   1:  PR[91,2] = PR[90,2] + 16.760;
   1:L PR[91] R[100]mm/sec CNT100;
   1:  PR[91,1] = PR[90,1] + -20.956;
   1:  PR[91,2] = PR[90,2] + 17.044;
   1:L PR[91] R[100]mm/sec CNT100;
   1:  PR[91,1] = PR[90,1] + -22.141;
   1:  PR[91,2] = PR[90,2] + 17.148;
   1:L PR[91] R[100]mm/sec CNT100;
   1:  PR[91,1] = PR[90,1] + -24.744;
   1:  PR[91,2] = PR[90,2] + 17.432;
   1:L PR[91] R[100]mm/sec CNT100;
   1:  PR[91,1] = PR[90,1] + -25.936;
   1:  PR[91,2] = PR[90,2] + 17.327;
   1:L PR[91] R[100]mm/sec CNT100;
   1:  PR[91,1] = PR[90,1] + -28.415;
   1:  PR[91,2] = PR[90,2] + 17.040;
   1:L PR[91] R[100]mm/sec CNT100;
   1:  PR[91,1] = PR[90,1] + -29.641;
   1:  PR[91,2] = PR[90,2] + 16.711;
   1:L PR[91] R[100]mm/sec CNT100;
   1:  PR[91,1] = PR[90,1] + -31.889;
   1:  PR[91,2] = PR[90,2] + 15.918;
   1:L PR[91] R[100]mm/sec CNT100;
   1:  PR[91,1] = PR[90,1] + -33.097;
   1:  PR[91,2] = PR[90,2] + 15.354;
   1:L PR[91] R[100]mm/sec CNT100;
   1:  PR[91,1] = PR[90,1] + -35.033;
   1:  PR[91,2] = PR[90,2] + 14.131;
   1:L PR[91] R[100]mm/sec CNT100;
   1:  PR[91,1] = PR[90,1] + -36.169;
   1:  PR[91,2] = PR[90,2] + 13.336;
   1:L PR[91] R[100]mm/sec CNT100;
   1:  PR[91,1] = PR[90,1] + -38.779;
   1:  PR[91,2] = PR[90,2] + 10.719;
   1:L PR[91] R[100]mm/sec CNT100TB   .50sec,CALL END_PUD;
   1:  PR[92] = PR[91];
   1:  PR[92,3] = PR[92,3] + 20;
   1:J PR[92] 10% FINE;
   1:  PR[91,1] = PR[90,1] + -69.247;
   1:  PR[91,2] = PR[90,2] + 16.551;
   1:  PR[92] = PR[91];
   1:  PR[92,3] = PR[92,3] + 20;
   1:J PR[92] 10% FINE;
   1:L PR[91] R[100]mm/sec CNT100;
   1:  CALL LASER_DRAHT_START;
   1:  PR[91,1] = PR[90,1] + -72.638;
   1:  PR[91,2] = PR[90,2] + 17.266;
   1:L PR[91] R[100]mm/sec CNT100;
   1:  PR[91,1] = PR[90,1] + -73.009;
   1:  PR[91,2] = PR[90,2] + 17.298;
   1:L PR[91] R[100]mm/sec CNT100;
   1:  PR[91,1] = PR[90,1] + -76.253;
   1:  PR[91,2] = PR[90,2] + 17.293;
   1:L PR[91] R[100]mm/sec CNT100;
   1:  PR[91,1] = PR[90,1] + -76.771;
   1:  PR[91,2] = PR[90,2] + 17.248;
   1:L PR[91] R[100]mm/sec CNT100;
   1:  PR[91,1] = PR[90,1] + -79.751;
   1:  PR[91,2] = PR[90,2] + 16.609;
   1:L PR[91] R[100]mm/sec CNT100;
   1:  PR[91,1] = PR[90,1] + -80.365;
   1:  PR[91,2] = PR[90,2] + 16.445;
   1:L PR[91] R[100]mm/sec CNT100;
   1:  PR[91,1] = PR[90,1] + -81.001;
   1:  PR[91,2] = PR[90,2] + 16.148;
   1:L PR[91] R[100]mm/sec CNT100;
   1:  PR[91,1] = PR[90,1] + -83.731;
   1:  PR[91,2] = PR[90,2] + 14.925;
   1:L PR[91] R[100]mm/sec CNT100;
   1:  PR[91,1] = PR[90,1] + -84.359;
   1:  PR[91,2] = PR[90,2] + 14.485;
   1:L PR[91] R[100]mm/sec CNT100;
   1:  PR[91,1] = PR[90,1] + -86.653;
   1:  PR[91,2] = PR[90,2] + 12.813;
   1:L PR[91] R[100]mm/sec CNT100;
   1:  PR[91,1] = PR[90,1] + -87.257;
   1:  PR[91,2] = PR[90,2] + 12.209;
   1:L PR[91] R[100]mm/sec CNT100;
   1:  PR[91,1] = PR[90,1] + -89.073;
   1:  PR[91,2] = PR[90,2] + 10.188;
   1:L PR[91] R[100]mm/sec CNT100;
   1:  PR[91,1] = PR[90,1] + -89.607;
   1:  PR[91,2] = PR[90,2] + 9.426;
   1:L PR[91] R[100]mm/sec CNT100;
   1:  PR[91,1] = PR[90,1] + -90.920;
   1:  PR[91,2] = PR[90,2] + 7.148;
   1:L PR[91] R[100]mm/sec CNT100;
   1:  PR[91,1] = PR[90,1] + -91.333;
   1:  PR[91,2] = PR[90,2] + 6.263;
   1:L PR[91] R[100]mm/sec CNT100;
   1:  PR[91,1] = PR[90,1] + -92.127;
   1:  PR[91,2] = PR[90,2] + 3.815;
   1:L PR[91] R[100]mm/sec CNT100;
   1:  PR[91,1] = PR[90,1] + -92.384;
   1:  PR[91,2] = PR[90,2] + 2.855;
   1:L PR[91] R[100]mm/sec CNT100;
   1:  PR[91,1] = PR[90,1] + -92.476;
   1:  PR[91,2] = PR[90,2] + 1.801;
   1:L PR[91] R[100]mm/sec CNT100;
   1:  PR[91,1] = PR[90,1] + -92.743;
   1:  PR[91,2] = PR[90,2] + -0.747;
   1:L PR[91] R[100]mm/sec CNT100;
   1:  PR[91,1] = PR[90,1] + -92.665;
   1:  PR[91,2] = PR[90,2] + -1.630;
   1:L PR[91] R[100]mm/sec CNT100;
   1:  PR[91,1] = PR[90,1] + -92.614;
   1:  PR[91,2] = PR[90,2] + -1.837;
   1:L PR[91] R[100]mm/sec CNT100;
   1:  PR[91,1] = PR[90,1] + -92.361;
   1:  PR[91,2] = PR[90,2] + -4.254;
   1:L PR[91] R[100]mm/sec CNT100;
   1:  PR[91,1] = PR[90,1] + -92.040;
   1:  PR[91,2] = PR[90,2] + -5.451;
   1:L PR[91] R[100]mm/sec CNT100;
   1:  PR[91,1] = PR[90,1] + -91.331;
   1:  PR[91,2] = PR[90,2] + -7.640;
   1:L PR[91] R[100]mm/sec CNT100;
   1:  PR[91,1] = PR[90,1] + -90.820;
   1:  PR[91,2] = PR[90,2] + -8.736;
   1:L PR[91] R[100]mm/sec CNT100;
   1:  PR[91,1] = PR[90,1] + -89.646;
   1:  PR[91,2] = PR[90,2] + -10.772;
   1:L PR[91] R[100]mm/sec CNT100;
   1:  PR[91,1] = PR[90,1] + -88.976;
   1:  PR[91,2] = PR[90,2] + -11.729;
   1:L PR[91] R[100]mm/sec CNT100;
   1:  PR[91,1] = PR[90,1] + -87.353;
   1:  PR[91,2] = PR[90,2] + -13.536;
   1:L PR[91] R[100]mm/sec CNT100;
   1:  PR[91,1] = PR[90,1] + -86.576;
   1:  PR[91,2] = PR[90,2] + -14.313;
   1:L PR[91] R[100]mm/sec CNT100;
   1:  PR[91,1] = PR[90,1] + -84.525;
   1:  PR[91,2] = PR[90,2] + -15.809;
   1:L PR[91] R[100]mm/sec CNT100;
   1:  PR[91,1] = PR[90,1] + -83.677;
   1:  PR[91,2] = PR[90,2] + -16.402;
   1:L PR[91] R[100]mm/sec CNT100;
   1:  PR[91,1] = PR[90,1] + -82.739;
   1:  PR[91,2] = PR[90,2] + -16.839;
   1:L PR[91] R[100]mm/sec CNT100;
   1:  PR[91,1] = PR[90,1] + -80.387;
   1:  PR[91,2] = PR[90,2] + -17.893;
   1:L PR[91] R[100]mm/sec CNT100;
   1:  PR[91,1] = PR[90,1] + -79.501;
   1:  PR[91,2] = PR[90,2] + -18.130;
   1:L PR[91] R[100]mm/sec CNT100;
   1:  PR[91,1] = PR[90,1] + -76.834;
   1:  PR[91,2] = PR[90,2] + -18.703;
   1:L PR[91] R[100]mm/sec CNT100;
   1:  PR[91,1] = PR[90,1] + -76.040;
   1:  PR[91,2] = PR[90,2] + -18.772;
   1:L PR[91] R[100]mm/sec CNT100;
   1:  PR[91,1] = PR[90,1] + -73.135;
   1:  PR[91,2] = PR[90,2] + -18.779;
   1:L PR[91] R[100]mm/sec CNT100;
   1:  PR[91,1] = PR[90,1] + -72.474;
   1:  PR[91,2] = PR[90,2] + -18.721;
   1:L PR[91] R[100]mm/sec CNT100;
   1:  PR[91,1] = PR[90,1] + -69.435;
   1:  PR[91,2] = PR[90,2] + -18.082;
   1:L PR[91] R[100]mm/sec CNT100;
   1:  PR[91,1] = PR[90,1] + -68.955;
   1:  PR[91,2] = PR[90,2] + -17.954;
   1:L PR[91] R[100]mm/sec CNT100;
   1:  PR[91,1] = PR[90,1] + -68.437;
   1:  PR[91,2] = PR[90,2] + -17.712;
   1:L PR[91] R[100]mm/sec CNT100;
   1:  PR[91,1] = PR[90,1] + -65.552;
   1:  PR[91,2] = PR[90,2] + -16.440;
   1:L PR[91] R[100]mm/sec CNT100;
   1:  PR[91,1] = PR[90,1] + -62.499;
   1:  PR[91,2] = PR[90,2] + -14.245;
   1:L PR[91] R[100]mm/sec CNT100;
   1:  PR[91,1] = PR[90,1] + -62.350;
   1:  PR[91,2] = PR[90,2] + -14.095;
   1:L PR[91] R[100]mm/sec CNT100;
   1:  PR[91,1] = PR[90,1] + -59.945;
   1:  PR[91,2] = PR[90,2] + -11.434;
   1:L PR[91] R[100]mm/sec CNT100;
   1:  PR[91,1] = PR[90,1] + -59.899;
   1:  PR[91,2] = PR[90,2] + -11.367;
   1:L PR[91] R[100]mm/sec CNT100;
   1:  PR[91,1] = PR[90,1] + -58.021;
   1:  PR[91,2] = PR[90,2] + -8.128;
   1:L PR[91] R[100]mm/sec CNT100;
   1:  PR[91,1] = PR[90,1] + -56.846;
   1:  PR[91,2] = PR[90,2] + -4.503;
   1:L PR[91] R[100]mm/sec CNT100;
   1:  PR[91,1] = PR[90,1] + -56.756;
   1:  PR[91,2] = PR[90,2] + -3.498;
   1:L PR[91] R[100]mm/sec CNT100;
   1:  PR[91,1] = PR[90,1] + -56.459;
   1:  PR[91,2] = PR[90,2] + -0.724;
   1:L PR[91] R[100]mm/sec CNT100;
   1:  PR[91,1] = PR[90,1] + -56.811;
   1:  PR[91,2] = PR[90,2] + 2.748;
   1:L PR[91] R[100]mm/sec CNT100;
   1:  PR[91,1] = PR[90,1] + -56.836;
   1:  PR[91,2] = PR[90,2] + 3.070;
   1:L PR[91] R[100]mm/sec CNT100;
   1:  PR[91,1] = PR[90,1] + -58.024;
   1:  PR[91,2] = PR[90,2] + 6.648;
   1:L PR[91] R[100]mm/sec CNT100;
   1:  PR[91,1] = PR[90,1] + -59.962;
   1:  PR[91,2] = PR[90,2] + 9.930;
   1:L PR[91] R[100]mm/sec CNT100;
   1:  PR[91,1] = PR[90,1] + -62.542;
   1:  PR[91,2] = PR[90,2] + 12.758;
   1:L PR[91] R[100]mm/sec CNT100;
   1:  PR[91,1] = PR[90,1] + -65.608;
   1:  PR[91,2] = PR[90,2] + 14.970;
   1:L PR[91] R[100]mm/sec CNT100;
   1:  PR[91,1] = PR[90,1] + -69.045;
   1:  PR[91,2] = PR[90,2] + 16.497;
   1:L PR[91] R[100]mm/sec CNT100;
   1:  PR[91,1] = PR[90,1] + -69.247;
   1:  PR[91,2] = PR[90,2] + 16.551;
   1:L PR[91] R[100]mm/sec CNT100TB   .50sec,CALL END_PUD;
   1:  PR[92] = PR[91];
   1:  PR[92,3] = PR[92,3] + 20;
   1:J PR[92] 10% FINE;
   1:  PR[91] = PR[90];
   1:  PR[91,1] = PR[90,1] + 39.926;
   1:  PR[91,2] = PR[90,2] + -10.972;
   1:  PR[91,3] = PR[90,3] + 17.095;
   1:  PR[92] = PR[91];
   1:  PR[92,3] = PR[92,3] + 20;
   1:J PR[92] 10% FINE;
   1:L PR[91] R[100]mm/sec CNT100;
   1:  CALL LASER_DRAHT_START;
   1:  PR[91,1] = PR[90,1] + 40.681;
   1:  PR[91,2] = PR[90,2] + -9.894;
   1:L PR[91] R[100]mm/sec CNT100;
   1:  PR[91,1] = PR[90,1] + 41.235;
   1:  PR[91,2] = PR[90,2] + -8.707;
   1:L PR[91] R[100]mm/sec CNT100;
   1:  PR[91,1] = PR[90,1] + 42.319;
   1:  PR[91,2] = PR[90,2] + -6.084;
   1:L PR[91] R[100]mm/sec CNT100;
   1:  PR[91,1] = PR[90,1] + 42.639;
   1:  PR[91,2] = PR[90,2] + -4.891;
   1:L PR[91] R[100]mm/sec CNT100;
   1:  PR[91,1] = PR[90,1] + 42.760;
   1:  PR[91,2] = PR[90,2] + -3.506;
   1:L PR[91] R[100]mm/sec CNT100;
   1:  PR[91,1] = PR[90,1] + 43.087;
   1:  PR[91,2] = PR[90,2] + -0.700;
   1:L PR[91] R[100]mm/sec CNT100;
   1:  PR[91,1] = PR[90,1] + 43.018;
   1:  PR[91,2] = PR[90,2] + 0.088;
   1:L PR[91] R[100]mm/sec CNT100;
   1:  PR[91,1] = PR[90,1] + 43.010;
   1:  PR[91,2] = PR[90,2] + 0.654;
   1:L PR[91] R[100]mm/sec CNT100;
   1:  PR[91,1] = PR[90,1] + 42.650;
   1:  PR[91,2] = PR[90,2] + 3.390;
   1:L PR[91] R[100]mm/sec CNT100;
   1:  PR[91,1] = PR[90,1] + 42.319;
   1:  PR[91,2] = PR[90,2] + 4.626;
   1:L PR[91] R[100]mm/sec CNT100;
   1:  PR[91,1] = PR[90,1] + 41.234;
   1:  PR[91,2] = PR[90,2] + 7.249;
   1:L PR[91] R[100]mm/sec CNT100;
   1:  PR[91,1] = PR[90,1] + 40.680;
   1:  PR[91,2] = PR[90,2] + 8.436;
   1:L PR[91] R[100]mm/sec CNT100;
   1:  PR[91,1] = PR[90,1] + 39.925;
   1:  PR[91,2] = PR[90,2] + 9.514;
   1:L PR[91] R[100]mm/sec CNT100;
   1:  PR[91,1] = PR[90,1] + 38.193;
   1:  PR[91,2] = PR[90,2] + 11.777;
   1:L PR[91] R[100]mm/sec CNT100;
   1:  PR[91,1] = PR[90,1] + 37.306;
   1:  PR[91,2] = PR[90,2] + 12.663;
   1:L PR[91] R[100]mm/sec CNT100;
   1:  PR[91,1] = PR[90,1] + 35.023;
   1:  PR[91,2] = PR[90,2] + 14.420;
   1:L PR[91] R[100]mm/sec CNT100;
   1:  PR[91,1] = PR[90,1] + 33.972;
   1:  PR[91,2] = PR[90,2] + 15.155;
   1:L PR[91] R[100]mm/sec CNT100;
   1:  PR[91,1] = PR[90,1] + 32.809;
   1:  PR[91,2] = PR[90,2] + 15.697;
   1:L PR[91] R[100]mm/sec CNT100;
   1:  PR[91,1] = PR[90,1] + 30.132;
   1:  PR[91,2] = PR[90,2] + 16.810;
   1:L PR[91] R[100]mm/sec CNT100;
   1:  PR[91,1] = PR[90,1] + 28.953;
   1:  PR[91,2] = PR[90,2] + 17.126;
   1:L PR[91] R[100]mm/sec CNT100;
   1:  PR[91,1] = PR[90,1] + 26.036;
   1:  PR[91,2] = PR[90,2] + 17.515;
   1:L PR[91] R[100]mm/sec CNT100;
   1:  PR[91,1] = PR[90,1] + 24.803;
   1:  PR[91,2] = PR[90,2] + 17.623;
   1:L PR[91] R[100]mm/sec CNT100;
   1:  PR[91,1] = PR[90,1] + 23.566;
   1:  PR[91,2] = PR[90,2] + 17.514;
   1:L PR[91] R[100]mm/sec CNT100;
   1:  PR[91,1] = PR[90,1] + 20.624;
   1:  PR[91,2] = PR[90,2] + 17.131;
   1:L PR[91] R[100]mm/sec CNT100;
   1:  PR[91,1] = PR[90,1] + 19.533;
   1:  PR[91,2] = PR[90,2] + 16.839;
   1:L PR[91] R[100]mm/sec CNT100;
   1:  PR[91,1] = PR[90,1] + 18.350;
   1:  PR[91,2] = PR[90,2] + 16.287;
   1:L PR[91] R[100]mm/sec CNT100;
   1:  PR[91,1] = PR[90,1] + 15.586;
   1:  PR[91,2] = PR[90,2] + 15.148;
   1:L PR[91] R[100]mm/sec CNT100;
   1:  PR[91,1] = PR[90,1] + 14.640;
   1:  PR[91,2] = PR[90,2] + 14.486;
   1:L PR[91] R[100]mm/sec CNT100;
   1:  PR[91,1] = PR[90,1] + 12.231;
   1:  PR[91,2] = PR[90,2] + 12.643;
   1:L PR[91] R[100]mm/sec CNT100;
   1:  PR[91,1] = PR[90,1] + 11.430;
   1:  PR[91,2] = PR[90,2] + 11.843;
   1:L PR[91] R[100]mm/sec CNT100;
   1:  PR[91,1] = PR[90,1] + 9.561;
   1:  PR[91,2] = PR[90,2] + 9.411;
   1:L PR[91] R[100]mm/sec CNT100;
   1:  PR[91,1] = PR[90,1] + 8.892;
   1:  PR[91,2] = PR[90,2] + 8.456;
   1:L PR[91] R[100]mm/sec CNT100;
   1:  PR[91,1] = PR[90,1] + 8.401;
   1:  PR[91,2] = PR[90,2] + 7.402;
   1:L PR[91] R[100]mm/sec CNT100;
   1:  PR[91,1] = PR[90,1] + 7.220;
   1:  PR[91,2] = PR[90,2] + 4.557;
   1:L PR[91] R[100]mm/sec CNT100;
   1:  PR[91,1] = PR[90,1] + 6.944;
   1:  PR[91,2] = PR[90,2] + 3.525;
   1:L PR[91] R[100]mm/sec CNT100;
   1:  PR[91,1] = PR[90,1] + 6.836;
   1:  PR[91,2] = PR[90,2] + 2.291;
   1:L PR[91] R[100]mm/sec CNT100;
   1:  PR[91,1] = PR[90,1] + 6.437;
   1:  PR[91,2] = PR[90,2] + -0.772;
   1:L PR[91] R[100]mm/sec CNT100;
   1:  PR[91,1] = PR[90,1] + 6.545;
   1:  PR[91,2] = PR[90,2] + -2.003;
   1:L PR[91] R[100]mm/sec CNT100;
   1:  PR[91,1] = PR[90,1] + 6.932;
   1:  PR[91,2] = PR[90,2] + -4.941;
   1:L PR[91] R[100]mm/sec CNT100;
   1:  PR[91,1] = PR[90,1] + 7.221;
   1:  PR[91,2] = PR[90,2] + -6.017;
   1:L PR[91] R[100]mm/sec CNT100;
   1:  PR[91,1] = PR[90,1] + 8.401;
   1:  PR[91,2] = PR[90,2] + -8.861;
   1:L PR[91] R[100]mm/sec CNT100;
   1:  PR[91,1] = PR[90,1] + 8.893;
   1:  PR[91,2] = PR[90,2] + -9.916;
   1:L PR[91] R[100]mm/sec CNT100;
   1:  PR[91,1] = PR[90,1] + 9.562;
   1:  PR[91,2] = PR[90,2] + -10.871;
   1:L PR[91] R[100]mm/sec CNT100;
   1:  PR[91,1] = PR[90,1] + 11.432;
   1:  PR[91,2] = PR[90,2] + -13.303;
   1:L PR[91] R[100]mm/sec CNT100;
   1:  PR[91,1] = PR[90,1] + 12.233;
   1:  PR[91,2] = PR[90,2] + -14.104;
   1:L PR[91] R[100]mm/sec CNT100;
   1:  PR[91,1] = PR[90,1] + 14.642;
   1:  PR[91,2] = PR[90,2] + -15.947;
   1:L PR[91] R[100]mm/sec CNT100;
   1:  PR[91,1] = PR[90,1] + 15.626;
   1:  PR[91,2] = PR[90,2] + -16.635;
   1:L PR[91] R[100]mm/sec CNT100;
   1:  PR[91,1] = PR[90,1] + 16.708;
   1:  PR[91,2] = PR[90,2] + -17.139;
   1:L PR[91] R[100]mm/sec CNT100;
   1:  PR[91,1] = PR[90,1] + 19.492;
   1:  PR[91,2] = PR[90,2] + -18.287;
   1:L PR[91] R[100]mm/sec CNT100;
   1:  PR[91,1] = PR[90,1] + 20.629;
   1:  PR[91,2] = PR[90,2] + -18.591;
   1:L PR[91] R[100]mm/sec CNT100;
   1:  PR[91,1] = PR[90,1] + 23.571;
   1:  PR[91,2] = PR[90,2] + -18.974;
   1:L PR[91] R[100]mm/sec CNT100;
   1:  PR[91,1] = PR[90,1] + 24.807;
   1:  PR[91,2] = PR[90,2] + -19.082;
   1:L PR[91] R[100]mm/sec CNT100;
   1:  PR[91,1] = PR[90,1] + 26.041;
   1:  PR[91,2] = PR[90,2] + -18.973;
   1:L PR[91] R[100]mm/sec CNT100;
   1:  PR[91,1] = PR[90,1] + 28.958;
   1:  PR[91,2] = PR[90,2] + -18.584;
   1:L PR[91] R[100]mm/sec CNT100;
   1:  PR[91,1] = PR[90,1] + 30.095;
   1:  PR[91,2] = PR[90,2] + -18.279;
   1:L PR[91] R[100]mm/sec CNT100;
   1:  PR[91,1] = PR[90,1] + 31.314;
   1:  PR[91,2] = PR[90,2] + -17.710;
   1:L PR[91] R[100]mm/sec CNT100;
   1:  PR[91,1] = PR[90,1] + 34.009;
   1:  PR[91,2] = PR[90,2] + -16.588;
   1:L PR[91] R[100]mm/sec CNT100;
   1:  PR[91,1] = PR[90,1] + 35.025;
   1:  PR[91,2] = PR[90,2] + -15.877;
   1:L PR[91] R[100]mm/sec CNT100;
   1:  PR[91,1] = PR[90,1] + 37.309;
   1:  PR[91,2] = PR[90,2] + -14.120;
   1:L PR[91] R[100]mm/sec CNT100;
   1:  PR[91,1] = PR[90,1] + 38.194;
   1:  PR[91,2] = PR[90,2] + -13.235;
   1:L PR[91] R[100]mm/sec CNT100;
   1:  PR[91,1] = PR[90,1] + 39.926;
   1:  PR[91,2] = PR[90,2] + -10.972;
   1:L PR[91] R[100]mm/sec CNT100TB   .50sec,CALL END_PUD;
   1:  PR[92] = PR[91];
   1:  PR[92,3] = PR[92,3] + 20;
   1:J PR[92] 10% FINE;
   1:  PR[91,1] = PR[90,1] + 66.363;
   1:  PR[91,2] = PR[90,2] + -17.228;
   1:  PR[92] = PR[91];
   1:  PR[92,3] = PR[92,3] + 20;
   1:J PR[92] 10% FINE;
   1:L PR[91] R[100]mm/sec CNT100;
   1:  CALL LASER_DRAHT_START;
   1:  PR[91,1] = PR[90,1] + 70.322;
   1:  PR[91,2] = PR[90,2] + -18.536;
   1:L PR[91] R[100]mm/sec CNT100;
   1:  PR[91,1] = PR[90,1] + 74.437;
   1:  PR[91,2] = PR[90,2] + -18.969;
   1:L PR[91] R[100]mm/sec CNT100;
   1:  PR[91,1] = PR[90,1] + 78.453;
   1:  PR[91,2] = PR[90,2] + -18.498;
   1:L PR[91] R[100]mm/sec CNT100;
   1:  PR[91,1] = PR[90,1] + 78.574;
   1:  PR[91,2] = PR[90,2] + -18.466;
   1:L PR[91] R[100]mm/sec CNT100;
   1:  PR[91,1] = PR[90,1] + 82.168;
   1:  PR[91,2] = PR[90,2] + -17.196;
   1:L PR[91] R[100]mm/sec CNT100;
   1:  PR[91,1] = PR[90,1] + 82.426;
   1:  PR[91,2] = PR[90,2] + -17.075;
   1:L PR[91] R[100]mm/sec CNT100;
   1:  PR[91,1] = PR[90,1] + 85.451;
   1:  PR[91,2] = PR[90,2] + -15.161;
   1:L PR[91] R[100]mm/sec CNT100;
   1:  PR[91,1] = PR[90,1] + 85.794;
   1:  PR[91,2] = PR[90,2] + -14.921;
   1:L PR[91] R[100]mm/sec CNT100;
   1:  PR[91,1] = PR[90,1] + 88.596;
   1:  PR[91,2] = PR[90,2] + -12.106;
   1:L PR[91] R[100]mm/sec CNT100;
   1:  PR[91,1] = PR[90,1] + 88.895;
   1:  PR[91,2] = PR[90,2] + -11.679;
   1:L PR[91] R[100]mm/sec CNT100;
   1:  PR[91,1] = PR[90,1] + 90.676;
   1:  PR[91,2] = PR[90,2] + -8.834;
   1:L PR[91] R[100]mm/sec CNT100;
   1:  PR[91,1] = PR[90,1] + 90.926;
   1:  PR[91,2] = PR[90,2] + -8.298;
   1:L PR[91] R[100]mm/sec CNT100;
   1:  PR[91,1] = PR[90,1] + 91.999;
   1:  PR[91,2] = PR[90,2] + -5.217;
   1:L PR[91] R[100]mm/sec CNT100;
   1:  PR[91,1] = PR[90,1] + 92.158;
   1:  PR[91,2] = PR[90,2] + -4.626;
   1:L PR[91] R[100]mm/sec CNT100;
   1:  PR[91,1] = PR[90,1] + 92.219;
   1:  PR[91,2] = PR[90,2] + -3.924;
   1:L PR[91] R[100]mm/sec CNT100;
   1:  PR[91,1] = PR[90,1] + 92.576;
   1:  PR[91,2] = PR[90,2] + -0.706;
   1:L PR[91] R[100]mm/sec CNT100;
   1:  PR[91,1] = PR[90,1] + 92.516;
   1:  PR[91,2] = PR[90,2] + -0.019;
   1:L PR[91] R[100]mm/sec CNT100;
   1:  PR[91,1] = PR[90,1] + 92.164;
   1:  PR[91,2] = PR[90,2] + 3.145;
   1:L PR[91] R[100]mm/sec CNT100;
   1:  PR[91,1] = PR[90,1] + 92.000;
   1:  PR[91,2] = PR[90,2] + 3.757;
   1:L PR[91] R[100]mm/sec CNT100;
   1:  PR[91,1] = PR[90,1] + 90.926;
   1:  PR[91,2] = PR[90,2] + 6.839;
   1:L PR[91] R[100]mm/sec CNT100;
   1:  PR[91,1] = PR[90,1] + 90.676;
   1:  PR[91,2] = PR[90,2] + 7.374;
   1:L PR[91] R[100]mm/sec CNT100;
   1:  PR[91,1] = PR[90,1] + 88.895;
   1:  PR[91,2] = PR[90,2] + 10.220;
   1:L PR[91] R[100]mm/sec CNT100;
   1:  PR[91,1] = PR[90,1] + 88.596;
   1:  PR[91,2] = PR[90,2] + 10.646;
   1:L PR[91] R[100]mm/sec CNT100;
   1:  PR[91,1] = PR[90,1] + 85.795;
   1:  PR[91,2] = PR[90,2] + 13.461;
   1:L PR[91] R[100]mm/sec CNT100;
   1:  PR[91,1] = PR[90,1] + 85.452;
   1:  PR[91,2] = PR[90,2] + 13.702;
   1:L PR[91] R[100]mm/sec CNT100;
   1:  PR[91,1] = PR[90,1] + 82.427;
   1:  PR[91,2] = PR[90,2] + 15.616;
   1:L PR[91] R[100]mm/sec CNT100;
   1:  PR[91,1] = PR[90,1] + 82.169;
   1:  PR[91,2] = PR[90,2] + 15.736;
   1:L PR[91] R[100]mm/sec CNT100;
   1:  PR[91,1] = PR[90,1] + 78.575;
   1:  PR[91,2] = PR[90,2] + 17.007;
   1:L PR[91] R[100]mm/sec CNT100;
   1:  PR[91,1] = PR[90,1] + 78.454;
   1:  PR[91,2] = PR[90,2] + 17.039;
   1:L PR[91] R[100]mm/sec CNT100;
   1:  PR[91,1] = PR[90,1] + 74.404;
   1:  PR[91,2] = PR[90,2] + 17.509;
   1:L PR[91] R[100]mm/sec CNT100;
   1:  PR[91,1] = PR[90,1] + 70.322;
   1:  PR[91,2] = PR[90,2] + 17.077;
   1:L PR[91] R[100]mm/sec CNT100;
   1:  PR[91,1] = PR[90,1] + 66.363;
   1:  PR[91,2] = PR[90,2] + 15.770;
   1:L PR[91] R[100]mm/sec CNT100;
   1:  PR[91,1] = PR[90,1] + 62.797;
   1:  PR[91,2] = PR[90,2] + 13.627;
   1:L PR[91] R[100]mm/sec CNT100;
   1:  PR[91,1] = PR[90,1] + 60.309;
   1:  PR[91,2] = PR[90,2] + 11.224;
   1:L PR[91] R[100]mm/sec CNT100;
   1:  PR[91,1] = PR[90,1] + 59.790;
   1:  PR[91,2] = PR[90,2] + 10.737;
   1:L PR[91] R[100]mm/sec CNT100;
   1:  PR[91,1] = PR[90,1] + 57.527;
   1:  PR[91,2] = PR[90,2] + 7.273;
   1:L PR[91] R[100]mm/sec CNT100;
   1:  PR[91,1] = PR[90,1] + 56.112;
   1:  PR[91,2] = PR[90,2] + 3.380;
   1:L PR[91] R[100]mm/sec CNT100;
   1:  PR[91,1] = PR[90,1] + 55.793;
   1:  PR[91,2] = PR[90,2] + 0.666;
   1:L PR[91] R[100]mm/sec CNT100;
   1:  PR[91,1] = PR[90,1] + 55.791;
   1:  PR[91,2] = PR[90,2] + 0.069;
   1:L PR[91] R[100]mm/sec CNT100;
   1:  PR[91,1] = PR[90,1] + 55.695;
   1:  PR[91,2] = PR[90,2] + -0.750;
   1:L PR[91] R[100]mm/sec CNT100;
   1:  PR[91,1] = PR[90,1] + 55.965;
   1:  PR[91,2] = PR[90,2] + -3.567;
   1:L PR[91] R[100]mm/sec CNT100;
   1:  PR[91,1] = PR[90,1] + 56.113;
   1:  PR[91,2] = PR[90,2] + -4.840;
   1:L PR[91] R[100]mm/sec CNT100;
   1:  PR[91,1] = PR[90,1] + 57.527;
   1:  PR[91,2] = PR[90,2] + -8.732;
   1:L PR[91] R[100]mm/sec CNT100;
   1:  PR[91,1] = PR[90,1] + 59.798;
   1:  PR[91,2] = PR[90,2] + -12.207;
   1:L PR[91] R[100]mm/sec CNT100;
   1:  PR[91,1] = PR[90,1] + 62.356;
   1:  PR[91,2] = PR[90,2] + -14.674;
   1:L PR[91] R[100]mm/sec CNT100;
   1:  PR[91,1] = PR[90,1] + 62.787;
   1:  PR[91,2] = PR[90,2] + -15.080;
   1:L PR[91] R[100]mm/sec CNT100;
   1:  PR[91,1] = PR[90,1] + 66.363;
   1:  PR[91,2] = PR[90,2] + -17.228;
   1:L PR[91] R[100]mm/sec CNT100TB   .50sec,CALL END_PUD;
   1:  PR[92] = PR[91];
   1:  PR[92,3] = PR[92,3] + 20;
   1:J PR[92] 10% FINE;
   1:  PR[91,1] = PR[90,1] + -35.228;
   1:  PR[91,2] = PR[90,2] + 13.987;
   1:  PR[92] = PR[91];
   1:  PR[92,3] = PR[92,3] + 20;
   1:J PR[92] 10% FINE;
   1:L PR[91] R[100]mm/sec CNT100;
   1:  CALL LASER_DRAHT_START;
   1:  PR[91,1] = PR[90,1] + -36.084;
   1:  PR[91,2] = PR[90,2] + 13.387;
   1:L PR[91] R[100]mm/sec CNT100;
   1:  PR[91,1] = PR[90,1] + -38.765;
   1:  PR[91,2] = PR[90,2] + 10.698;
   1:L PR[91] R[100]mm/sec CNT100;
   1:  PR[91,1] = PR[90,1] + -39.394;
   1:  PR[91,2] = PR[90,2] + 9.800;
   1:L PR[91] R[100]mm/sec CNT100;
   1:  PR[91,1] = PR[90,1] + -40.788;
   1:  PR[91,2] = PR[90,2] + 7.574;
   1:L PR[91] R[100]mm/sec CNT100;
   1:  PR[91,1] = PR[90,1] + -41.268;
   1:  PR[91,2] = PR[90,2] + 6.545;
   1:L PR[91] R[100]mm/sec CNT100;
   1:  PR[91,1] = PR[90,1] + -42.116;
   1:  PR[91,2] = PR[90,2] + 4.112;
   1:L PR[91] R[100]mm/sec CNT100;
   1:  PR[91,1] = PR[90,1] + -42.409;
   1:  PR[91,2] = PR[90,2] + 3.018;
   1:L PR[91] R[100]mm/sec CNT100;
   1:  PR[91,1] = PR[90,1] + -42.516;
   1:  PR[91,2] = PR[90,2] + 1.794;
   1:L PR[91] R[100]mm/sec CNT100;
   1:  PR[91,1] = PR[90,1] + -42.803;
   1:  PR[91,2] = PR[90,2] + -0.754;
   1:L PR[91] R[100]mm/sec CNT100;
   1:  PR[91,1] = PR[90,1] + -42.701;
   1:  PR[91,2] = PR[90,2] + -1.915;
   1:L PR[91] R[100]mm/sec CNT100;
   1:  PR[91,1] = PR[90,1] + -42.416;
   1:  PR[91,2] = PR[90,2] + -4.453;
   1:L PR[91] R[100]mm/sec CNT100;
   1:  PR[91,1] = PR[90,1] + -42.117;
   1:  PR[91,2] = PR[90,2] + -5.570;
   1:L PR[91] R[100]mm/sec CNT100;
   1:  PR[91,1] = PR[90,1] + -41.268;
   1:  PR[91,2] = PR[90,2] + -8.004;
   1:L PR[91] R[100]mm/sec CNT100;
   1:  PR[91,1] = PR[90,1] + -40.789;
   1:  PR[91,2] = PR[90,2] + -9.032;
   1:L PR[91] R[100]mm/sec CNT100;
   1:  PR[91,1] = PR[90,1] + -39.394;
   1:  PR[91,2] = PR[90,2] + -11.258;
   1:L PR[91] R[100]mm/sec CNT100;
   1:  PR[91,1] = PR[90,1] + -38.766;
   1:  PR[91,2] = PR[90,2] + -12.156;
   1:L PR[91] R[100]mm/sec CNT100;
   1:  PR[91,1] = PR[90,1] + -36.085;
   1:  PR[91,2] = PR[90,2] + -14.846;
   1:L PR[91] R[100]mm/sec CNT100;
   1:  PR[91,1] = PR[90,1] + -35.228;
   1:  PR[91,2] = PR[90,2] + -15.446;
   1:L PR[91] R[100]mm/sec CNT100;
   1:  PR[91,1] = PR[90,1] + -32.913;
   1:  PR[91,2] = PR[90,2] + -16.908;
   1:L PR[91] R[100]mm/sec CNT100;
   1:  PR[91,1] = PR[90,1] + -32.023;
   1:  PR[91,2] = PR[90,2] + -17.324;
   1:L PR[91] R[100]mm/sec CNT100;
   1:  PR[91,1] = PR[90,1] + -29.336;
   1:  PR[91,2] = PR[90,2] + -18.271;
   1:L PR[91] R[100]mm/sec CNT100;
   1:  PR[91,1] = PR[90,1] + -28.488;
   1:  PR[91,2] = PR[90,2] + -18.499;
   1:L PR[91] R[100]mm/sec CNT100;
   1:  PR[91,1] = PR[90,1] + -27.506;
   1:  PR[91,2] = PR[90,2] + -18.585;
   1:L PR[91] R[100]mm/sec CNT100;
   1:  PR[91,1] = PR[90,1] + -24.631;
   1:  PR[91,2] = PR[90,2] + -18.921;
   1:L PR[91] R[100]mm/sec CNT100;
   1:  PR[91,1] = PR[90,1] + -23.815;
   1:  PR[91,2] = PR[90,2] + -18.849;
   1:L PR[91] R[100]mm/sec CNT100;
   1:  PR[91,1] = PR[90,1] + -20.798;
   1:  PR[91,2] = PR[90,2] + -18.519;
   1:L PR[91] R[100]mm/sec CNT100;
   1:  PR[91,1] = PR[90,1] + -20.096;
   1:  PR[91,2] = PR[90,2] + -18.330;
   1:L PR[91] R[100]mm/sec CNT100;
   1:  PR[91,1] = PR[90,1] + -17.087;
   1:  PR[91,2] = PR[90,2] + -17.288;
   1:L PR[91] R[100]mm/sec CNT100;
   1:  PR[91,1] = PR[90,1] + -16.513;
   1:  PR[91,2] = PR[90,2] + -17.020;
   1:L PR[91] R[100]mm/sec CNT100;
   1:  PR[91,1] = PR[90,1] + -13.688;
   1:  PR[91,2] = PR[90,2] + -15.255;
   1:L PR[91] R[100]mm/sec CNT100;
   1:  PR[91,1] = PR[90,1] + -13.244;
   1:  PR[91,2] = PR[90,2] + -14.945;
   1:L PR[91] R[100]mm/sec CNT100;
   1:  PR[91,1] = PR[90,1] + -10.425;
   1:  PR[91,2] = PR[90,2] + -12.139;
   1:L PR[91] R[100]mm/sec CNT100;
   1:  PR[91,1] = PR[90,1] + -10.161;
   1:  PR[91,2] = PR[90,2] + -11.761;
   1:L PR[91] R[100]mm/sec CNT100;
   1:  PR[91,1] = PR[90,1] + -8.289;
   1:  PR[91,2] = PR[90,2] + -8.796;
   1:L PR[91] R[100]mm/sec CNT100;
   1:  PR[91,1] = PR[90,1] + -8.121;
   1:  PR[91,2] = PR[90,2] + -8.436;
   1:L PR[91] R[100]mm/sec CNT100;
   1:  PR[91,1] = PR[90,1] + -6.932;
   1:  PR[91,2] = PR[90,2] + -5.047;
   1:L PR[91] R[100]mm/sec CNT100;
   1:  PR[91,1] = PR[90,1] + -6.843;
   1:  PR[91,2] = PR[90,2] + -4.713;
   1:L PR[91] R[100]mm/sec CNT100;
   1:  PR[91,1] = PR[90,1] + -6.435;
   1:  PR[91,2] = PR[90,2] + -0.715;
   1:L PR[91] R[100]mm/sec CNT100;
   1:  PR[91,1] = PR[90,1] + -6.473;
   1:  PR[91,2] = PR[90,2] + -0.283;
   1:L PR[91] R[100]mm/sec CNT100;
   1:  PR[91,1] = PR[90,1] + -6.456;
   1:  PR[91,2] = PR[90,2] + -0.150;
   1:L PR[91] R[100]mm/sec CNT100;
   1:  PR[91,1] = PR[90,1] + -6.840;
   1:  PR[91,2] = PR[90,2] + 3.243;
   1:L PR[91] R[100]mm/sec CNT100;
   1:  PR[91,1] = PR[90,1] + -6.932;
   1:  PR[91,2] = PR[90,2] + 3.588;
   1:L PR[91] R[100]mm/sec CNT100;
   1:  PR[91,1] = PR[90,1] + -8.121;
   1:  PR[91,2] = PR[90,2] + 6.977;
   1:L PR[91] R[100]mm/sec CNT100;
   1:  PR[91,1] = PR[90,1] + -8.289;
   1:  PR[91,2] = PR[90,2] + 7.337;
   1:L PR[91] R[100]mm/sec CNT100;
   1:  PR[91,1] = PR[90,1] + -10.161;
   1:  PR[91,2] = PR[90,2] + 10.302;
   1:L PR[91] R[100]mm/sec CNT100;
   1:  PR[91,1] = PR[90,1] + -10.425;
   1:  PR[91,2] = PR[90,2] + 10.680;
   1:L PR[91] R[100]mm/sec CNT100;
   1:  PR[91,1] = PR[90,1] + -13.244;
   1:  PR[91,2] = PR[90,2] + 13.486;
   1:L PR[91] R[100]mm/sec CNT100;
   1:  PR[91,1] = PR[90,1] + -13.687;
   1:  PR[91,2] = PR[90,2] + 13.796;
   1:L PR[91] R[100]mm/sec CNT100;
   1:  PR[91,1] = PR[90,1] + -16.513;
   1:  PR[91,2] = PR[90,2] + 15.561;
   1:L PR[91] R[100]mm/sec CNT100;
   1:  PR[91,1] = PR[90,1] + -17.087;
   1:  PR[91,2] = PR[90,2] + 15.829;
   1:L PR[91] R[100]mm/sec CNT100;
   1:  PR[91,1] = PR[90,1] + -20.095;
   1:  PR[91,2] = PR[90,2] + 16.871;
   1:L PR[91] R[100]mm/sec CNT100;
   1:  PR[91,1] = PR[90,1] + -20.777;
   1:  PR[91,2] = PR[90,2] + 17.054;
   1:L PR[91] R[100]mm/sec CNT100;
   1:  PR[91,1] = PR[90,1] + -21.573;
   1:  PR[91,2] = PR[90,2] + 17.124;
   1:L PR[91] R[100]mm/sec CNT100;
   1:  PR[91,1] = PR[90,1] + -24.681;
   1:  PR[91,2] = PR[90,2] + 17.463;
   1:L PR[91] R[100]mm/sec CNT100;
   1:  PR[91,1] = PR[90,1] + -25.498;
   1:  PR[91,2] = PR[90,2] + 17.391;
   1:L PR[91] R[100]mm/sec CNT100;
   1:  PR[91,1] = PR[90,1] + -28.460;
   1:  PR[91,2] = PR[90,2] + 17.047;
   1:L PR[91] R[100]mm/sec CNT100;
   1:  PR[91,1] = PR[90,1] + -29.335;
   1:  PR[91,2] = PR[90,2] + 16.813;
   1:L PR[91] R[100]mm/sec CNT100;
   1:  PR[91,1] = PR[90,1] + -32.023;
   1:  PR[91,2] = PR[90,2] + 15.865;
   1:L PR[91] R[100]mm/sec CNT100;
   1:  PR[91,1] = PR[90,1] + -32.913;
   1:  PR[91,2] = PR[90,2] + 15.450;
   1:L PR[91] R[100]mm/sec CNT100;
   1:  PR[91,1] = PR[90,1] + -35.228;
   1:  PR[91,2] = PR[90,2] + 13.987;
   1:L PR[91] R[100]mm/sec CNT100TB   .50sec,CALL END_PUD;
   1:  PR[92] = PR[91];
   1:  PR[92,3] = PR[92,3] + 20;
   1:J PR[92] 10% FINE;
   1:  PR[91,1] = PR[90,1] + -89.407;
   1:  PR[91,2] = PR[90,2] + 9.650;
   1:  PR[92] = PR[91];
   1:  PR[92,3] = PR[92,3] + 20;
   1:J PR[92] 10% FINE;
   1:L PR[91] R[100]mm/sec CNT100;
   1:  CALL LASER_DRAHT_START;
   1:  PR[91,1] = PR[90,1] + -90.976;
   1:  PR[91,2] = PR[90,2] + 6.931;
   1:L PR[91] R[100]mm/sec CNT100;
   1:  PR[91,1] = PR[90,1] + -91.212;
   1:  PR[91,2] = PR[90,2] + 6.424;
   1:L PR[91] R[100]mm/sec CNT100;
   1:  PR[91,1] = PR[90,1] + -92.160;
   1:  PR[91,2] = PR[90,2] + 3.500;
   1:L PR[91] R[100]mm/sec CNT100;
   1:  PR[91,1] = PR[90,1] + -92.310;
   1:  PR[91,2] = PR[90,2] + 2.940;
   1:L PR[91] R[100]mm/sec CNT100;
   1:  PR[91,1] = PR[90,1] + -92.366;
   1:  PR[91,2] = PR[90,2] + 2.296;
   1:L PR[91] R[100]mm/sec CNT100;
   1:  PR[91,1] = PR[90,1] + -92.684;
   1:  PR[91,2] = PR[90,2] + -0.747;
   1:L PR[91] R[100]mm/sec CNT100;
   1:  PR[91,1] = PR[90,1] + -92.643;
   1:  PR[91,2] = PR[90,2] + -1.223;
   1:L PR[91] R[100]mm/sec CNT100;
   1:  PR[91,1] = PR[90,1] + -92.581;
   1:  PR[91,2] = PR[90,2] + -1.471;
   1:L PR[91] R[100]mm/sec CNT100;
   1:  PR[91,1] = PR[90,1] + -92.282;
   1:  PR[91,2] = PR[90,2] + -4.331;
   1:L PR[91] R[100]mm/sec CNT100;
   1:  PR[91,1] = PR[90,1] + -92.057;
   1:  PR[91,2] = PR[90,2] + -5.169;
   1:L PR[91] R[100]mm/sec CNT100;
   1:  PR[91,1] = PR[90,1] + -91.210;
   1:  PR[91,2] = PR[90,2] + -7.786;
   1:L PR[91] R[100]mm/sec CNT100;
   1:  PR[91,1] = PR[90,1] + -90.857;
   1:  PR[91,2] = PR[90,2] + -8.541;
   1:L PR[91] R[100]mm/sec CNT100;
   1:  PR[91,1] = PR[90,1] + -89.454;
   1:  PR[91,2] = PR[90,2] + -10.975;
   1:L PR[91] R[100]mm/sec CNT100;
   1:  PR[91,1] = PR[90,1] + -89.005;
   1:  PR[91,2] = PR[90,2] + -11.616;
   1:L PR[91] R[100]mm/sec CNT100;
   1:  PR[91,1] = PR[90,1] + -87.066;
   1:  PR[91,2] = PR[90,2] + -13.777;
   1:L PR[91] R[100]mm/sec CNT100;
   1:  PR[91,1] = PR[90,1] + -86.568;
   1:  PR[91,2] = PR[90,2] + -14.274;
   1:L PR[91] R[100]mm/sec CNT100;
   1:  PR[91,1] = PR[90,1] + -84.118;
   1:  PR[91,2] = PR[90,2] + -16.061;
   1:L PR[91] R[100]mm/sec CNT100;
   1:  PR[91,1] = PR[90,1] + -83.617;
   1:  PR[91,2] = PR[90,2] + -16.411;
   1:L PR[91] R[100]mm/sec CNT100;
   1:  PR[91,1] = PR[90,1] + -80.230;
   1:  PR[91,2] = PR[90,2] + -17.941;
   1:L PR[91] R[100]mm/sec CNT100;
   1:  PR[91,1] = PR[90,1] + -79.762;
   1:  PR[91,2] = PR[90,2] + -18.066;
   1:L PR[91] R[100]mm/sec CNT100;
   1:  PR[91,1] = PR[90,1] + -76.579;
   1:  PR[91,2] = PR[90,2] + -18.750;
   1:L PR[91] R[100]mm/sec CNT100;
   1:  PR[91,1] = PR[90,1] + -76.234;
   1:  PR[91,2] = PR[90,2] + -18.780;
   1:L PR[91] R[100]mm/sec CNT100;
   1:  PR[91,1] = PR[90,1] + -72.768;
   1:  PR[91,2] = PR[90,2] + -18.788;
   1:L PR[91] R[100]mm/sec CNT100;
   1:  PR[91,1] = PR[90,1] + -72.581;
   1:  PR[91,2] = PR[90,2] + -18.771;
   1:L PR[91] R[100]mm/sec CNT100;
   1:  PR[91,1] = PR[90,1] + -68.958;
   1:  PR[91,2] = PR[90,2] + -18.010;
   1:L PR[91] R[100]mm/sec CNT100;
   1:  PR[91,1] = PR[90,1] + -68.944;
   1:  PR[91,2] = PR[90,2] + -18.006;
   1:L PR[91] R[100]mm/sec CNT100;
   1:  PR[91,1] = PR[90,1] + -65.452;
   1:  PR[91,2] = PR[90,2] + -16.462;
   1:L PR[91] R[100]mm/sec CNT100;
   1:  PR[91,1] = PR[90,1] + -62.314;
   1:  PR[91,2] = PR[90,2] + -14.239;
   1:L PR[91] R[100]mm/sec CNT100;
   1:  PR[91,1] = PR[90,1] + -59.704;
   1:  PR[91,2] = PR[90,2] + -11.424;
   1:L PR[91] R[100]mm/sec CNT100;
   1:  PR[91,1] = PR[90,1] + -57.750;
   1:  PR[91,2] = PR[90,2] + -8.136;
   1:L PR[91] R[100]mm/sec CNT100;
   1:  PR[91,1] = PR[90,1] + -56.542;
   1:  PR[91,2] = PR[90,2] + -4.517;
   1:L PR[91] R[100]mm/sec CNT100;
   1:  PR[91,1] = PR[90,1] + -56.190;
   1:  PR[91,2] = PR[90,2] + -1.263;
   1:L PR[91] R[100]mm/sec CNT100;
   1:  PR[91,1] = PR[90,1] + -56.176;
   1:  PR[91,2] = PR[90,2] + -0.799;
   1:L PR[91] R[100]mm/sec CNT100;
   1:  PR[91,1] = PR[90,1] + -56.396;
   1:  PR[91,2] = PR[90,2] + 1.423;
   1:L PR[91] R[100]mm/sec CNT100;
   1:  PR[91,1] = PR[90,1] + -56.419;
   1:  PR[91,2] = PR[90,2] + 2.134;
   1:L PR[91] R[100]mm/sec CNT100;
   1:  PR[91,1] = PR[90,1] + -56.519;
   1:  PR[91,2] = PR[90,2] + 3.061;
   1:L PR[91] R[100]mm/sec CNT100;
   1:  PR[91,1] = PR[90,1] + -57.723;
   1:  PR[91,2] = PR[90,2] + 6.683;
   1:L PR[91] R[100]mm/sec CNT100;
   1:  PR[91,1] = PR[90,1] + -59.672;
   1:  PR[91,2] = PR[90,2] + 9.973;
   1:L PR[91] R[100]mm/sec CNT100;
   1:  PR[91,1] = PR[90,1] + -62.271;
   1:  PR[91,2] = PR[90,2] + 12.789;
   1:L PR[91] R[100]mm/sec CNT100;
   1:  PR[91,1] = PR[90,1] + -65.408;
   1:  PR[91,2] = PR[90,2] + 15.006;
   1:L PR[91] R[100]mm/sec CNT100;
   1:  PR[91,1] = PR[90,1] + -68.940;
   1:  PR[91,2] = PR[90,2] + 16.531;
   1:L PR[91] R[100]mm/sec CNT100;
   1:  PR[91,1] = PR[90,1] + -72.681;
   1:  PR[91,2] = PR[90,2] + 17.298;
   1:L PR[91] R[100]mm/sec CNT100;
   1:  PR[91,1] = PR[90,1] + -76.484;
   1:  PR[91,2] = PR[90,2] + 17.297;
   1:L PR[91] R[100]mm/sec CNT100;
   1:  PR[91,1] = PR[90,1] + -76.502;
   1:  PR[91,2] = PR[90,2] + 17.295;
   1:L PR[91] R[100]mm/sec CNT100;
   1:  PR[91,1] = PR[90,1] + -80.055;
   1:  PR[91,2] = PR[90,2] + 16.535;
   1:L PR[91] R[100]mm/sec CNT100;
   1:  PR[91,1] = PR[90,1] + -80.222;
   1:  PR[91,2] = PR[90,2] + 16.490;
   1:L PR[91] R[100]mm/sec CNT100;
   1:  PR[91,1] = PR[90,1] + -83.652;
   1:  PR[91,2] = PR[90,2] + 14.947;
   1:L PR[91] R[100]mm/sec CNT100;
   1:  PR[91,1] = PR[90,1] + -86.660;
   1:  PR[91,2] = PR[90,2] + 12.766;
   1:L PR[91] R[100]mm/sec CNT100;
   1:  PR[91,1] = PR[90,1] + -86.952;
   1:  PR[91,2] = PR[90,2] + 12.474;
   1:L PR[91] R[100]mm/sec CNT100;
   1:  PR[91,1] = PR[90,1] + -89.119;
   1:  PR[91,2] = PR[90,2] + 10.062;
   1:L PR[91] R[100]mm/sec CNT100;
   1:  PR[91,1] = PR[90,1] + -89.407;
   1:  PR[91,2] = PR[90,2] + 9.650;
   1:L PR[91] R[100]mm/sec CNT100TB   .50sec,CALL END_PUD;
   1:  PR[92] = PR[91];
   1:  PR[92,3] = PR[92,3] + 20;
   1:J PR[92] 10% FINE;
   1:  PR[91] = PR[90];
   1:  PR[91,1] = PR[90,1] + 7.095;
   1:  PR[91,2] = PR[90,2] + -5.877;
   1:  PR[91,3] = PR[90,3] + 18.395;
   1:  PR[92] = PR[91];
   1:  PR[92,3] = PR[92,3] + 20;
   1:J PR[92] 10% FINE;
   1:L PR[91] R[100]mm/sec CNT100;
   1:  CALL LASER_DRAHT_START;
   1:  PR[91,1] = PR[90,1] + 8.468;
   1:  PR[91,2] = PR[90,2] + -9.184;
   1:L PR[91] R[100]mm/sec CNT100;
   1:  PR[91,1] = PR[90,1] + 8.823;
   1:  PR[91,2] = PR[90,2] + -9.945;
   1:L PR[91] R[100]mm/sec CNT100;
   1:  PR[91,1] = PR[90,1] + 9.306;
   1:  PR[91,2] = PR[90,2] + -10.635;
   1:L PR[91] R[100]mm/sec CNT100;
   1:  PR[91,1] = PR[90,1] + 11.480;
   1:  PR[91,2] = PR[90,2] + -13.462;
   1:L PR[91] R[100]mm/sec CNT100;
   1:  PR[91,1] = PR[90,1] + 12.054;
   1:  PR[91,2] = PR[90,2] + -14.036;
   1:L PR[91] R[100]mm/sec CNT100;
   1:  PR[91,1] = PR[90,1] + 14.855;
   1:  PR[91,2] = PR[90,2] + -16.179;
   1:L PR[91] R[100]mm/sec CNT100;
   1:  PR[91,1] = PR[90,1] + 15.577;
   1:  PR[91,2] = PR[90,2] + -16.684;
   1:L PR[91] R[100]mm/sec CNT100;
   1:  PR[91,1] = PR[90,1] + 16.371;
   1:  PR[91,2] = PR[90,2] + -17.054;
   1:L PR[91] R[100]mm/sec CNT100;
   1:  PR[91,1] = PR[90,1] + 19.609;
   1:  PR[91,2] = PR[90,2] + -18.389;
   1:L PR[91] R[100]mm/sec CNT100;
   1:  PR[91,1] = PR[90,1] + 20.440;
   1:  PR[91,2] = PR[90,2] + -18.611;
   1:L PR[91] R[100]mm/sec CNT100;
   1:  PR[91,1] = PR[90,1] + 23.862;
   1:  PR[91,2] = PR[90,2] + -19.056;
   1:L PR[91] R[100]mm/sec CNT100;
   1:  PR[91,1] = PR[90,1] + 24.787;
   1:  PR[91,2] = PR[90,2] + -19.137;
   1:L PR[91] R[100]mm/sec CNT100;
   1:  PR[91,1] = PR[90,1] + 25.710;
   1:  PR[91,2] = PR[90,2] + -19.056;
   1:L PR[91] R[100]mm/sec CNT100;
   1:  PR[91,1] = PR[90,1] + 29.104;
   1:  PR[91,2] = PR[90,2] + -18.603;
   1:L PR[91] R[100]mm/sec CNT100;
   1:  PR[91,1] = PR[90,1] + 29.942;
   1:  PR[91,2] = PR[90,2] + -18.378;
   1:L PR[91] R[100]mm/sec CNT100;
   1:  PR[91,1] = PR[90,1] + 30.882;
   1:  PR[91,2] = PR[90,2] + -17.939;
   1:L PR[91] R[100]mm/sec CNT100;
   1:  PR[91,1] = PR[90,1] + 34.017;
   1:  PR[91,2] = PR[90,2] + -16.634;
   1:L PR[91] R[100]mm/sec CNT100;
   1:  PR[91,1] = PR[90,1] + 34.782;
   1:  PR[91,2] = PR[90,2] + -16.098;
   1:L PR[91] R[100]mm/sec CNT100;
   1:  PR[91,1] = PR[90,1] + 37.438;
   1:  PR[91,2] = PR[90,2] + -14.055;
   1:L PR[91] R[100]mm/sec CNT100;
   1:  PR[91,1] = PR[90,1] + 38.110;
   1:  PR[91,2] = PR[90,2] + -13.384;
   1:L PR[91] R[100]mm/sec CNT100;
   1:  PR[91,1] = PR[90,1] + 40.126;
   1:  PR[91,2] = PR[90,2] + -10.751;
   1:L PR[91] R[100]mm/sec CNT100;
   1:  PR[91,1] = PR[90,1] + 40.707;
   1:  PR[91,2] = PR[90,2] + -9.920;
   1:L PR[91] R[100]mm/sec CNT100;
   1:  PR[91,1] = PR[90,1] + 41.133;
   1:  PR[91,2] = PR[90,2] + -9.006;
   1:L PR[91] R[100]mm/sec CNT100;
   1:  PR[91,1] = PR[90,1] + 42.395;
   1:  PR[91,2] = PR[90,2] + -5.954;
   1:L PR[91] R[100]mm/sec CNT100;
   1:  PR[91,1] = PR[90,1] + 42.637;
   1:  PR[91,2] = PR[90,2] + -5.051;
   1:L PR[91] R[100]mm/sec CNT100;
   1:  PR[91,1] = PR[90,1] + 42.732;
   1:  PR[91,2] = PR[90,2] + -3.965;
   1:L PR[91] R[100]mm/sec CNT100;
   1:  PR[91,1] = PR[90,1] + 43.113;
   1:  PR[91,2] = PR[90,2] + -0.700;
   1:L PR[91] R[100]mm/sec CNT100;
   1:  PR[91,1] = PR[90,1] + 43.078;
   1:  PR[91,2] = PR[90,2] + -0.305;
   1:L PR[91] R[100]mm/sec CNT100;
   1:  PR[91,1] = PR[90,1] + 43.068;
   1:  PR[91,2] = PR[90,2] + 0.355;
   1:L PR[91] R[100]mm/sec CNT100;
   1:  PR[91,1] = PR[90,1] + 42.648;
   1:  PR[91,2] = PR[90,2] + 3.550;
   1:L PR[91] R[100]mm/sec CNT100;
   1:  PR[91,1] = PR[90,1] + 42.395;
   1:  PR[91,2] = PR[90,2] + 4.496;
   1:L PR[91] R[100]mm/sec CNT100;
   1:  PR[91,1] = PR[90,1] + 41.133;
   1:  PR[91,2] = PR[90,2] + 7.548;
   1:L PR[91] R[100]mm/sec CNT100;
   1:  PR[91,1] = PR[90,1] + 40.707;
   1:  PR[91,2] = PR[90,2] + 8.462;
   1:L PR[91] R[100]mm/sec CNT100;
   1:  PR[91,1] = PR[90,1] + 40.124;
   1:  PR[91,2] = PR[90,2] + 9.293;
   1:L PR[91] R[100]mm/sec CNT100;
   1:  PR[91,1] = PR[90,1] + 38.109;
   1:  PR[91,2] = PR[90,2] + 11.926;
   1:L PR[91] R[100]mm/sec CNT100;
   1:  PR[91,1] = PR[90,1] + 37.437;
   1:  PR[91,2] = PR[90,2] + 12.598;
   1:L PR[91] R[100]mm/sec CNT100;
   1:  PR[91,1] = PR[90,1] + 34.781;
   1:  PR[91,2] = PR[90,2] + 14.641;
   1:L PR[91] R[100]mm/sec CNT100;
   1:  PR[91,1] = PR[90,1] + 33.980;
   1:  PR[91,2] = PR[90,2] + 15.201;
   1:L PR[91] R[100]mm/sec CNT100;
   1:  PR[91,1] = PR[90,1] + 33.095;
   1:  PR[91,2] = PR[90,2] + 15.613;
   1:L PR[91] R[100]mm/sec CNT100;
   1:  PR[91,1] = PR[90,1] + 29.980;
   1:  PR[91,2] = PR[90,2] + 16.909;
   1:L PR[91] R[100]mm/sec CNT100;
   1:  PR[91,1] = PR[90,1] + 29.100;
   1:  PR[91,2] = PR[90,2] + 17.145;
   1:L PR[91] R[100]mm/sec CNT100;
   1:  PR[91,1] = PR[90,1] + 25.707;
   1:  PR[91,2] = PR[90,2] + 17.598;
   1:L PR[91] R[100]mm/sec CNT100;
   1:  PR[91,1] = PR[90,1] + 24.784;
   1:  PR[91,2] = PR[90,2] + 17.678;
   1:L PR[91] R[100]mm/sec CNT100;
   1:  PR[91,1] = PR[90,1] + 23.858;
   1:  PR[91,2] = PR[90,2] + 17.597;
   1:L PR[91] R[100]mm/sec CNT100;
   1:  PR[91,1] = PR[90,1] + 20.436;
   1:  PR[91,2] = PR[90,2] + 17.152;
   1:L PR[91] R[100]mm/sec CNT100;
   1:  PR[91,1] = PR[90,1] + 19.650;
   1:  PR[91,2] = PR[90,2] + 16.941;
   1:L PR[91] R[100]mm/sec CNT100;
   1:  PR[91,1] = PR[90,1] + 18.753;
   1:  PR[91,2] = PR[90,2] + 16.522;
   1:L PR[91] R[100]mm/sec CNT100;
   1:  PR[91,1] = PR[90,1] + 15.538;
   1:  PR[91,2] = PR[90,2] + 15.198;
   1:L PR[91] R[100]mm/sec CNT100;
   1:  PR[91,1] = PR[90,1] + 14.854;
   1:  PR[91,2] = PR[90,2] + 14.719;
   1:L PR[91] R[100]mm/sec CNT100;
   1:  PR[91,1] = PR[90,1] + 12.052;
   1:  PR[91,2] = PR[90,2] + 12.576;
   1:L PR[91] R[100]mm/sec CNT100;
   1:  PR[91,1] = PR[90,1] + 11.479;
   1:  PR[91,2] = PR[90,2] + 12.003;
   1:L PR[91] R[100]mm/sec CNT100;
   1:  PR[91,1] = PR[90,1] + 9.305;
   1:  PR[91,2] = PR[90,2] + 9.175;
   1:L PR[91] R[100]mm/sec CNT100;
   1:  PR[91,1] = PR[90,1] + 8.823;
   1:  PR[91,2] = PR[90,2] + 8.486;
   1:L PR[91] R[100]mm/sec CNT100;
   1:  PR[91,1] = PR[90,1] + 8.468;
   1:  PR[91,2] = PR[90,2] + 7.724;
   1:L PR[91] R[100]mm/sec CNT100;
   1:  PR[91,1] = PR[90,1] + 7.095;
   1:  PR[91,2] = PR[90,2] + 4.417;
   1:L PR[91] R[100]mm/sec CNT100;
   1:  PR[91,1] = PR[90,1] + 6.903;
   1:  PR[91,2] = PR[90,2] + 3.700;
   1:L PR[91] R[100]mm/sec CNT100;
   1:  PR[91,1] = PR[90,1] + 6.823;
   1:  PR[91,2] = PR[90,2] + 2.789;
   1:L PR[91] R[100]mm/sec CNT100;
   1:  PR[91,1] = PR[90,1] + 6.360;
   1:  PR[91,2] = PR[90,2] + -0.772;
   1:L PR[91] R[100]mm/sec CNT100;
   1:  PR[91,1] = PR[90,1] + 6.441;
   1:  PR[91,2] = PR[90,2] + -1.698;
   1:L PR[91] R[100]mm/sec CNT100;
   1:  PR[91,1] = PR[90,1] + 6.892;
   1:  PR[91,2] = PR[90,2] + -5.116;
   1:L PR[91] R[100]mm/sec CNT100;
   1:  PR[91,1] = PR[90,1] + 7.095;
   1:  PR[91,2] = PR[90,2] + -5.877;
   1:L PR[91] R[100]mm/sec CNT100TB   .50sec,CALL END_PUD;
   1:  PR[92] = PR[91];
   1:  PR[92,3] = PR[92,3] + 20;
   1:J PR[92] 10% FINE;
   1:  PR[91,1] = PR[90,1] + 90.781;
   1:  PR[91,2] = PR[90,2] + -8.526;
   1:  PR[92] = PR[91];
   1:  PR[92,3] = PR[92,3] + 20;
   1:J PR[92] 10% FINE;
   1:L PR[91] R[100]mm/sec CNT100;
   1:  CALL LASER_DRAHT_START;
   1:  PR[91,1] = PR[90,1] + 92.029;
   1:  PR[91,2] = PR[90,2] + -4.945;
   1:L PR[91] R[100]mm/sec CNT100;
   1:  PR[91,1] = PR[90,1] + 92.087;
   1:  PR[91,2] = PR[90,2] + -4.726;
   1:L PR[91] R[100]mm/sec CNT100;
   1:  PR[91,1] = PR[90,1] + 92.523;
   1:  PR[91,2] = PR[90,2] + -0.708;
   1:L PR[91] R[100]mm/sec CNT100;
   1:  PR[91,1] = PR[90,1] + 92.497;
   1:  PR[91,2] = PR[90,2] + -0.414;
   1:L PR[91] R[100]mm/sec CNT100;
   1:  PR[91,1] = PR[90,1] + 92.088;
   1:  PR[91,2] = PR[90,2] + 3.264;
   1:L PR[91] R[100]mm/sec CNT100;
   1:  PR[91,1] = PR[90,1] + 92.029;
   1:  PR[91,2] = PR[90,2] + 3.486;
   1:L PR[91] R[100]mm/sec CNT100;
   1:  PR[91,1] = PR[90,1] + 90.781;
   1:  PR[91,2] = PR[90,2] + 7.067;
   1:L PR[91] R[100]mm/sec CNT100;
   1:  PR[91,1] = PR[90,1] + 90.705;
   1:  PR[91,2] = PR[90,2] + 7.230;
   1:L PR[91] R[100]mm/sec CNT100;
   1:  PR[91,1] = PR[90,1] + 88.635;
   1:  PR[91,2] = PR[90,2] + 10.536;
   1:L PR[91] R[100]mm/sec CNT100;
   1:  PR[91,1] = PR[90,1] + 88.579;
   1:  PR[91,2] = PR[90,2] + 10.617;
   1:L PR[91] R[100]mm/sec CNT100;
   1:  PR[91,1] = PR[90,1] + 85.719;
   1:  PR[91,2] = PR[90,2] + 13.493;
   1:L PR[91] R[100]mm/sec CNT100;
   1:  PR[91,1] = PR[90,1] + 82.268;
   1:  PR[91,2] = PR[90,2] + 15.686;
   1:L PR[91] R[100]mm/sec CNT100;
   1:  PR[91,1] = PR[90,1] + 78.355;
   1:  PR[91,2] = PR[90,2] + 17.082;
   1:L PR[91] R[100]mm/sec CNT100;
   1:  PR[91,1] = PR[90,1] + 74.216;
   1:  PR[91,2] = PR[90,2] + 17.593;
   1:L PR[91] R[100]mm/sec CNT100;
   1:  PR[91,1] = PR[90,1] + 70.055;
   1:  PR[91,2] = PR[90,2] + 17.188;
   1:L PR[91] R[100]mm/sec CNT100;
   1:  PR[91,1] = PR[90,1] + 66.870;
   1:  PR[91,2] = PR[90,2] + 16.132;
   1:L PR[91] R[100]mm/sec CNT100;
   1:  PR[91,1] = PR[90,1] + 66.062;
   1:  PR[91,2] = PR[90,2] + 15.878;
   1:L PR[91] R[100]mm/sec CNT100;
   1:  PR[91,1] = PR[90,1] + 63.495;
   1:  PR[91,2] = PR[90,2] + 14.328;
   1:L PR[91] R[100]mm/sec CNT100;
   1:  PR[91,1] = PR[90,1] + 62.465;
   1:  PR[91,2] = PR[90,2] + 13.727;
   1:L PR[91] R[100]mm/sec CNT100;
   1:  PR[91,1] = PR[90,1] + 60.556;
   1:  PR[91,2] = PR[90,2] + 11.884;
   1:L PR[91] R[100]mm/sec CNT100;
   1:  PR[91,1] = PR[90,1] + 59.438;
   1:  PR[91,2] = PR[90,2] + 10.834;
   1:L PR[91] R[100]mm/sec CNT100;
   1:  PR[91,1] = PR[90,1] + 58.166;
   1:  PR[91,2] = PR[90,2] + 8.875;
   1:L PR[91] R[100]mm/sec CNT100;
   1:  PR[91,1] = PR[90,1] + 57.142;
   1:  PR[91,2] = PR[90,2] + 7.334;
   1:L PR[91] R[100]mm/sec CNT100;
   1:  PR[91,1] = PR[90,1] + 55.712;
   1:  PR[91,2] = PR[90,2] + 3.416;
   1:L PR[91] R[100]mm/sec CNT100;
   1:  PR[91,1] = PR[90,1] + 55.503;
   1:  PR[91,2] = PR[90,2] + 1.632;
   1:L PR[91] R[100]mm/sec CNT100;
   1:  PR[91,1] = PR[90,1] + 55.501;
   1:  PR[91,2] = PR[90,2] + 1.218;
   1:L PR[91] R[100]mm/sec CNT100;
   1:  PR[91,1] = PR[90,1] + 55.271;
   1:  PR[91,2] = PR[90,2] + -0.750;
   1:L PR[91] R[100]mm/sec CNT100;
   1:  PR[91,1] = PR[90,1] + 55.447;
   1:  PR[91,2] = PR[90,2] + -2.581;
   1:L PR[91] R[100]mm/sec CNT100;
   1:  PR[91,1] = PR[90,1] + 55.713;
   1:  PR[91,2] = PR[90,2] + -4.876;
   1:L PR[91] R[100]mm/sec CNT100;
   1:  PR[91,1] = PR[90,1] + 57.145;
   1:  PR[91,2] = PR[90,2] + -8.803;
   1:L PR[91] R[100]mm/sec CNT100;
   1:  PR[91,1] = PR[90,1] + 58.377;
   1:  PR[91,2] = PR[90,2] + -10.698;
   1:L PR[91] R[100]mm/sec CNT100;
   1:  PR[91,1] = PR[90,1] + 59.438;
   1:  PR[91,2] = PR[90,2] + -12.297;
   1:L PR[91] R[100]mm/sec CNT100;
   1:  PR[91,1] = PR[90,1] + 61.324;
   1:  PR[91,2] = PR[90,2] + -14.115;
   1:L PR[91] R[100]mm/sec CNT100;
   1:  PR[91,1] = PR[90,1] + 62.465;
   1:  PR[91,2] = PR[90,2] + -15.190;
   1:L PR[91] R[100]mm/sec CNT100;
   1:  PR[91,1] = PR[90,1] + 65.061;
   1:  PR[91,2] = PR[90,2] + -16.755;
   1:L PR[91] R[100]mm/sec CNT100;
   1:  PR[91,1] = PR[90,1] + 66.062;
   1:  PR[91,2] = PR[90,2] + -17.340;
   1:L PR[91] R[100]mm/sec CNT100;
   1:  PR[91,1] = PR[90,1] + 69.339;
   1:  PR[91,2] = PR[90,2] + -18.423;
   1:L PR[91] R[100]mm/sec CNT100;
   1:  PR[91,1] = PR[90,1] + 70.041;
   1:  PR[91,2] = PR[90,2] + -18.645;
   1:L PR[91] R[100]mm/sec CNT100;
   1:  PR[91,1] = PR[90,1] + 74.216;
   1:  PR[91,2] = PR[90,2] + -19.051;
   1:L PR[91] R[100]mm/sec CNT100;
   1:  PR[91,1] = PR[90,1] + 78.355;
   1:  PR[91,2] = PR[90,2] + -18.540;
   1:L PR[91] R[100]mm/sec CNT100;
   1:  PR[91,1] = PR[90,1] + 82.268;
   1:  PR[91,2] = PR[90,2] + -17.145;
   1:L PR[91] R[100]mm/sec CNT100;
   1:  PR[91,1] = PR[90,1] + 85.718;
   1:  PR[91,2] = PR[90,2] + -14.952;
   1:L PR[91] R[100]mm/sec CNT100;
   1:  PR[91,1] = PR[90,1] + 88.578;
   1:  PR[91,2] = PR[90,2] + -12.076;
   1:L PR[91] R[100]mm/sec CNT100;
   1:  PR[91,1] = PR[90,1] + 88.635;
   1:  PR[91,2] = PR[90,2] + -11.995;
   1:L PR[91] R[100]mm/sec CNT100;
   1:  PR[91,1] = PR[90,1] + 90.705;
   1:  PR[91,2] = PR[90,2] + -8.689;
   1:L PR[91] R[100]mm/sec CNT100;
   1:  PR[91,1] = PR[90,1] + 90.781;
   1:  PR[91,2] = PR[90,2] + -8.526;
   1:L PR[91] R[100]mm/sec CNT100TB   .50sec,CALL END_PUD;
   1:  PR[92] = PR[91];
   1:  PR[92,3] = PR[92,3] + 20;
   1:J PR[92] 10% FINE;
   1:  PR[91,1] = PR[90,1] + -20.619;
   1:  PR[91,2] = PR[90,2] + -18.529;
   1:  PR[92] = PR[91];
   1:  PR[92,3] = PR[92,3] + 20;
   1:J PR[92] 10% FINE;
   1:L PR[91] R[100]mm/sec CNT100;
   1:  CALL LASER_DRAHT_START;
   1:  PR[91,1] = PR[90,1] + -20.293;
   1:  PR[91,2] = PR[90,2] + -18.441;
   1:L PR[91] R[100]mm/sec CNT100;
   1:  PR[91,1] = PR[90,1] + -16.796;
   1:  PR[91,2] = PR[90,2] + -17.230;
   1:L PR[91] R[100]mm/sec CNT100;
   1:  PR[91,1] = PR[90,1] + -16.589;
   1:  PR[91,2] = PR[90,2] + -17.133;
   1:L PR[91] R[100]mm/sec CNT100;
   1:  PR[91,1] = PR[90,1] + -13.305;
   1:  PR[91,2] = PR[90,2] + -15.082;
   1:L PR[91] R[100]mm/sec CNT100;
   1:  PR[91,1] = PR[90,1] + -13.204;
   1:  PR[91,2] = PR[90,2] + -15.011;
   1:L PR[91] R[100]mm/sec CNT100;
   1:  PR[91,1] = PR[90,1] + -10.293;
   1:  PR[91,2] = PR[90,2] + -12.116;
   1:L PR[91] R[100]mm/sec CNT100;
   1:  PR[91,1] = PR[90,1] + -10.276;
   1:  PR[91,2] = PR[90,2] + -12.091;
   1:L PR[91] R[100]mm/sec CNT100;
   1:  PR[91,1] = PR[90,1] + -8.112;
   1:  PR[91,2] = PR[90,2] + -8.663;
   1:L PR[91] R[100]mm/sec CNT100;
   1:  PR[91,1] = PR[90,1] + -6.761;
   1:  PR[91,2] = PR[90,2] + -4.814;
   1:L PR[91] R[100]mm/sec CNT100;
   1:  PR[91,1] = PR[90,1] + -6.470;
   1:  PR[91,2] = PR[90,2] + -1.992;
   1:L PR[91] R[100]mm/sec CNT100;
   1:  PR[91,1] = PR[90,1] + -6.310;
   1:  PR[91,2] = PR[90,2] + -0.613;
   1:L PR[91] R[100]mm/sec CNT100;
   1:  PR[91,1] = PR[90,1] + -6.754;
   1:  PR[91,2] = PR[90,2] + 3.304;
   1:L PR[91] R[100]mm/sec CNT100;
   1:  PR[91,1] = PR[90,1] + -8.113;
   1:  PR[91,2] = PR[90,2] + 7.205;
   1:L PR[91] R[100]mm/sec CNT100;
   1:  PR[91,1] = PR[90,1] + -10.276;
   1:  PR[91,2] = PR[90,2] + 10.632;
   1:L PR[91] R[100]mm/sec CNT100;
   1:  PR[91,1] = PR[90,1] + -10.293;
   1:  PR[91,2] = PR[90,2] + 10.657;
   1:L PR[91] R[100]mm/sec CNT100;
   1:  PR[91,1] = PR[90,1] + -13.204;
   1:  PR[91,2] = PR[90,2] + 13.552;
   1:L PR[91] R[100]mm/sec CNT100;
   1:  PR[91,1] = PR[90,1] + -13.305;
   1:  PR[91,2] = PR[90,2] + 13.623;
   1:L PR[91] R[100]mm/sec CNT100;
   1:  PR[91,1] = PR[90,1] + -16.589;
   1:  PR[91,2] = PR[90,2] + 15.674;
   1:L PR[91] R[100]mm/sec CNT100;
   1:  PR[91,1] = PR[90,1] + -16.796;
   1:  PR[91,2] = PR[90,2] + 15.771;
   1:L PR[91] R[100]mm/sec CNT100;
   1:  PR[91,1] = PR[90,1] + -20.293;
   1:  PR[91,2] = PR[90,2] + 16.982;
   1:L PR[91] R[100]mm/sec CNT100;
   1:  PR[91,1] = PR[90,1] + -20.597;
   1:  PR[91,2] = PR[90,2] + 17.064;
   1:L PR[91] R[100]mm/sec CNT100;
   1:  PR[91,1] = PR[90,1] + -21.004;
   1:  PR[91,2] = PR[90,2] + 17.100;
   1:L PR[91] R[100]mm/sec CNT100;
   1:  PR[91,1] = PR[90,1] + -24.618;
   1:  PR[91,2] = PR[90,2] + 17.494;
   1:L PR[91] R[100]mm/sec CNT100;
   1:  PR[91,1] = PR[90,1] + -25.060;
   1:  PR[91,2] = PR[90,2] + 17.455;
   1:L PR[91] R[100]mm/sec CNT100;
   1:  PR[91,1] = PR[90,1] + -28.504;
   1:  PR[91,2] = PR[90,2] + 17.055;
   1:L PR[91] R[100]mm/sec CNT100;
   1:  PR[91,1] = PR[90,1] + -29.030;
   1:  PR[91,2] = PR[90,2] + 16.914;
   1:L PR[91] R[100]mm/sec CNT100;
   1:  PR[91,1] = PR[90,1] + -32.156;
   1:  PR[91,2] = PR[90,2] + 15.812;
   1:L PR[91] R[100]mm/sec CNT100;
   1:  PR[91,1] = PR[90,1] + -32.728;
   1:  PR[91,2] = PR[90,2] + 15.545;
   1:L PR[91] R[100]mm/sec CNT100;
   1:  PR[91,1] = PR[90,1] + -35.422;
   1:  PR[91,2] = PR[90,2] + 13.843;
   1:L PR[91] R[100]mm/sec CNT100;
   1:  PR[91,1] = PR[90,1] + -35.999;
   1:  PR[91,2] = PR[90,2] + 13.439;
   1:L PR[91] R[100]mm/sec CNT100;
   1:  PR[91,1] = PR[90,1] + -38.751;
   1:  PR[91,2] = PR[90,2] + 10.677;
   1:L PR[91] R[100]mm/sec CNT100;
   1:  PR[91,1] = PR[90,1] + -39.189;
   1:  PR[91,2] = PR[90,2] + 10.051;
   1:L PR[91] R[100]mm/sec CNT100;
   1:  PR[91,1] = PR[90,1] + -40.812;
   1:  PR[91,2] = PR[90,2] + 7.460;
   1:L PR[91] R[100]mm/sec CNT100;
   1:  PR[91,1] = PR[90,1] + -41.153;
   1:  PR[91,2] = PR[90,2] + 6.729;
   1:L PR[91] R[100]mm/sec CNT100;
   1:  PR[91,1] = PR[90,1] + -42.142;
   1:  PR[91,2] = PR[90,2] + 3.895;
   1:L PR[91] R[100]mm/sec CNT100;
   1:  PR[91,1] = PR[90,1] + -42.351;
   1:  PR[91,2] = PR[90,2] + 3.115;
   1:L PR[91] R[100]mm/sec CNT100;
   1:  PR[91,1] = PR[90,1] + -42.429;
   1:  PR[91,2] = PR[90,2] + 2.213;
   1:L PR[91] R[100]mm/sec CNT100;
   1:  PR[91,1] = PR[90,1] + -42.763;
   1:  PR[91,2] = PR[90,2] + -0.754;
   1:L PR[91] R[100]mm/sec CNT100;
   1:  PR[91,1] = PR[90,1] + -42.690;
   1:  PR[91,2] = PR[90,2] + -1.595;
   1:L PR[91] R[100]mm/sec CNT100;
   1:  PR[91,1] = PR[90,1] + -42.357;
   1:  PR[91,2] = PR[90,2] + -4.549;
   1:L PR[91] R[100]mm/sec CNT100;
   1:  PR[91,1] = PR[90,1] + -42.142;
   1:  PR[91,2] = PR[90,2] + -5.354;
   1:L PR[91] R[100]mm/sec CNT100;
   1:  PR[91,1] = PR[90,1] + -41.154;
   1:  PR[91,2] = PR[90,2] + -8.187;
   1:L PR[91] R[100]mm/sec CNT100;
   1:  PR[91,1] = PR[90,1] + -40.813;
   1:  PR[91,2] = PR[90,2] + -8.919;
   1:L PR[91] R[100]mm/sec CNT100;
   1:  PR[91,1] = PR[90,1] + -39.189;
   1:  PR[91,2] = PR[90,2] + -11.510;
   1:L PR[91] R[100]mm/sec CNT100;
   1:  PR[91,1] = PR[90,1] + -38.752;
   1:  PR[91,2] = PR[90,2] + -12.135;
   1:L PR[91] R[100]mm/sec CNT100;
   1:  PR[91,1] = PR[90,1] + -36.000;
   1:  PR[91,2] = PR[90,2] + -14.897;
   1:L PR[91] R[100]mm/sec CNT100;
   1:  PR[91,1] = PR[90,1] + -35.422;
   1:  PR[91,2] = PR[90,2] + -15.302;
   1:L PR[91] R[100]mm/sec CNT100;
   1:  PR[91,1] = PR[90,1] + -32.728;
   1:  PR[91,2] = PR[90,2] + -17.004;
   1:L PR[91] R[100]mm/sec CNT100;
   1:  PR[91,1] = PR[90,1] + -32.156;
   1:  PR[91,2] = PR[90,2] + -17.271;
   1:L PR[91] R[100]mm/sec CNT100;
   1:  PR[91,1] = PR[90,1] + -29.030;
   1:  PR[91,2] = PR[90,2] + -18.373;
   1:L PR[91] R[100]mm/sec CNT100;
   1:  PR[91,1] = PR[90,1] + -28.532;
   1:  PR[91,2] = PR[90,2] + -18.506;
   1:L PR[91] R[100]mm/sec CNT100;
   1:  PR[91,1] = PR[90,1] + -27.913;
   1:  PR[91,2] = PR[90,2] + -18.561;
   1:L PR[91] R[100]mm/sec CNT100;
   1:  PR[91,1] = PR[90,1] + -24.568;
   1:  PR[91,2] = PR[90,2] + -18.952;
   1:L PR[91] R[100]mm/sec CNT100;
   1:  PR[91,1] = PR[90,1] + -24.127;
   1:  PR[91,2] = PR[90,2] + -18.913;
   1:L PR[91] R[100]mm/sec CNT100;
   1:  PR[91,1] = PR[90,1] + -20.619;
   1:  PR[91,2] = PR[90,2] + -18.529;
   1:L PR[91] R[100]mm/sec CNT100TB   .50sec,CALL END_PUD;
   1:  PR[92] = PR[91];
   1:  PR[92,3] = PR[92,3] + 20;
   1:J PR[92] 10% FINE;
   1:  PR[91,1] = PR[90,1] + -89.166;
   1:  PR[91,2] = PR[90,2] + 9.933;
   1:  PR[92] = PR[91];
   1:  PR[92,3] = PR[92,3] + 20;
   1:J PR[92] 10% FINE;
   1:L PR[91] R[100]mm/sec CNT100;
   1:  CALL LASER_DRAHT_START;
   1:  PR[91,1] = PR[90,1] + -89.207;
   1:  PR[91,2] = PR[90,2] + 9.874;
   1:L PR[91] R[100]mm/sec CNT100;
   1:  PR[91,1] = PR[90,1] + -91.031;
   1:  PR[91,2] = PR[90,2] + 6.713;
   1:L PR[91] R[100]mm/sec CNT100;
   1:  PR[91,1] = PR[90,1] + -91.091;
   1:  PR[91,2] = PR[90,2] + 6.585;
   1:L PR[91] R[100]mm/sec CNT100;
   1:  PR[91,1] = PR[90,1] + -92.193;
   1:  PR[91,2] = PR[90,2] + 3.185;
   1:L PR[91] R[100]mm/sec CNT100;
   1:  PR[91,1] = PR[90,1] + -92.240;
   1:  PR[91,2] = PR[90,2] + 3.009;
   1:L PR[91] R[100]mm/sec CNT100;
   1:  PR[91,1] = PR[90,1] + -92.627;
   1:  PR[91,2] = PR[90,2] + -0.745;
   1:L PR[91] R[100]mm/sec CNT100;
   1:  PR[91,1] = PR[90,1] + -92.620;
   1:  PR[91,2] = PR[90,2] + -0.816;
   1:L PR[91] R[100]mm/sec CNT100;
   1:  PR[91,1] = PR[90,1] + -92.549;
   1:  PR[91,2] = PR[90,2] + -1.104;
   1:L PR[91] R[100]mm/sec CNT100;
   1:  PR[91,1] = PR[90,1] + -92.203;
   1:  PR[91,2] = PR[90,2] + -4.407;
   1:L PR[91] R[100]mm/sec CNT100;
   1:  PR[91,1] = PR[90,1] + -92.075;
   1:  PR[91,2] = PR[90,2] + -4.886;
   1:L PR[91] R[100]mm/sec CNT100;
   1:  PR[91,1] = PR[90,1] + -91.088;
   1:  PR[91,2] = PR[90,2] + -7.932;
   1:L PR[91] R[100]mm/sec CNT100;
   1:  PR[91,1] = PR[90,1] + -90.895;
   1:  PR[91,2] = PR[90,2] + -8.346;
   1:L PR[91] R[100]mm/sec CNT100;
   1:  PR[91,1] = PR[90,1] + -89.262;
   1:  PR[91,2] = PR[90,2] + -11.178;
   1:L PR[91] R[100]mm/sec CNT100;
   1:  PR[91,1] = PR[90,1] + -89.034;
   1:  PR[91,2] = PR[90,2] + -11.504;
   1:L PR[91] R[100]mm/sec CNT100;
   1:  PR[91,1] = PR[90,1] + -86.778;
   1:  PR[91,2] = PR[90,2] + -14.017;
   1:L PR[91] R[100]mm/sec CNT100;
   1:  PR[91,1] = PR[90,1] + -86.562;
   1:  PR[91,2] = PR[90,2] + -14.233;
   1:L PR[91] R[100]mm/sec CNT100;
   1:  PR[91,1] = PR[90,1] + -83.533;
   1:  PR[91,2] = PR[90,2] + -16.433;
   1:L PR[91] R[100]mm/sec CNT100;
   1:  PR[91,1] = PR[90,1] + -80.077;
   1:  PR[91,2] = PR[90,2] + -17.988;
   1:L PR[91] R[100]mm/sec CNT100;
   1:  PR[91,1] = PR[90,1] + -80.023;
   1:  PR[91,2] = PR[90,2] + -18.002;
   1:L PR[91] R[100]mm/sec CNT100;
   1:  PR[91,1] = PR[90,1] + -76.403;
   1:  PR[91,2] = PR[90,2] + -18.780;
   1:L PR[91] R[100]mm/sec CNT100;
   1:  PR[91,1] = PR[90,1] + -72.528;
   1:  PR[91,2] = PR[90,2] + -18.805;
   1:L PR[91] R[100]mm/sec CNT100;
   1:  PR[91,1] = PR[90,1] + -68.729;
   1:  PR[91,2] = PR[90,2] + -18.043;
   1:L PR[91] R[100]mm/sec CNT100;
   1:  PR[91,1] = PR[90,1] + -65.171;
   1:  PR[91,2] = PR[90,2] + -16.520;
   1:L PR[91] R[100]mm/sec CNT100;
   1:  PR[91,1] = PR[90,1] + -62.008;
   1:  PR[91,2] = PR[90,2] + -14.300;
   1:L PR[91] R[100]mm/sec CNT100;
   1:  PR[91,1] = PR[90,1] + -59.384;
   1:  PR[91,2] = PR[90,2] + -11.476;
   1:L PR[91] R[100]mm/sec CNT100;
   1:  PR[91,1] = PR[90,1] + -57.416;
   1:  PR[91,2] = PR[90,2] + -8.174;
   1:L PR[91] R[100]mm/sec CNT100;
   1:  PR[91,1] = PR[90,1] + -56.199;
   1:  PR[91,2] = PR[90,2] + -4.538;
   1:L PR[91] R[100]mm/sec CNT100;
   1:  PR[91,1] = PR[90,1] + -55.929;
   1:  PR[91,2] = PR[90,2] + -2.039;
   1:L PR[91] R[100]mm/sec CNT100;
   1:  PR[91,1] = PR[90,1] + -55.893;
   1:  PR[91,2] = PR[90,2] + -0.799;
   1:L PR[91] R[100]mm/sec CNT100;
   1:  PR[91,1] = PR[90,1] + -55.977;
   1:  PR[91,2] = PR[90,2] + 0.049;
   1:L PR[91] R[100]mm/sec CNT100;
   1:  PR[91,1] = PR[90,1] + -56.016;
   1:  PR[91,2] = PR[90,2] + 1.277;
   1:L PR[91] R[100]mm/sec CNT100;
   1:  PR[91,1] = PR[90,1] + -56.211;
   1:  PR[91,2] = PR[90,2] + 3.080;
   1:L PR[91] R[100]mm/sec CNT100;
   1:  PR[91,1] = PR[90,1] + -57.423;
   1:  PR[91,2] = PR[90,2] + 6.718;
   1:L PR[91] R[100]mm/sec CNT100;
   1:  PR[91,1] = PR[90,1] + -59.384;
   1:  PR[91,2] = PR[90,2] + 10.021;
   1:L PR[91] R[100]mm/sec CNT100;
   1:  PR[91,1] = PR[90,1] + -61.998;
   1:  PR[91,2] = PR[90,2] + 12.846;
   1:L PR[91] R[100]mm/sec CNT100;
   1:  PR[91,1] = PR[90,1] + -65.150;
   1:  PR[91,2] = PR[90,2] + 15.068;
   1:L PR[91] R[100]mm/sec CNT100;
   1:  PR[91,1] = PR[90,1] + -68.697;
   1:  PR[91,2] = PR[90,2] + 16.594;
   1:L PR[91] R[100]mm/sec CNT100;
   1:  PR[91,1] = PR[90,1] + -72.483;
   1:  PR[91,2] = PR[90,2] + 17.358;
   1:L PR[91] R[100]mm/sec CNT100;
   1:  PR[91,1] = PR[90,1] + -76.341;
   1:  PR[91,2] = PR[90,2] + 17.331;
   1:L PR[91] R[100]mm/sec CNT100;
   1:  PR[91,1] = PR[90,1] + -80.104;
   1:  PR[91,2] = PR[90,2] + 16.518;
   1:L PR[91] R[100]mm/sec CNT100;
   1:  PR[91,1] = PR[90,1] + -83.588;
   1:  PR[91,2] = PR[90,2] + 14.961;
   1:L PR[91] R[100]mm/sec CNT100;
   1:  PR[91,1] = PR[90,1] + -86.622;
   1:  PR[91,2] = PR[90,2] + 12.752;
   1:L PR[91] R[100]mm/sec CNT100;
   1:  PR[91,1] = PR[90,1] + -89.166;
   1:  PR[91,2] = PR[90,2] + 9.933;
   1:L PR[91] R[100]mm/sec CNT100TB   .50sec,CALL END_PUD;
   1:  PR[92] = PR[91];
   1:  PR[92,3] = PR[92,3] + 20;
   1:J PR[92] 10% FINE;
   1:  PR[91] = PR[90];
   1:  PR[91,1] = PR[90,1] + 11.874;
   1:  PR[91,2] = PR[90,2] + -13.968;
   1:  PR[91,3] = PR[90,3] + 19.695;
   1:  PR[92] = PR[91];
   1:  PR[92,3] = PR[92,3] + 20;
   1:J PR[92] 10% FINE;
   1:L PR[91] R[100]mm/sec CNT100;
   1:  CALL LASER_DRAHT_START;
   1:  PR[91,1] = PR[90,1] + 15.068;
   1:  PR[91,2] = PR[90,2] + -16.411;
   1:L PR[91] R[100]mm/sec CNT100;
   1:  PR[91,1] = PR[90,1] + 15.529;
   1:  PR[91,2] = PR[90,2] + -16.733;
   1:L PR[91] R[100]mm/sec CNT100;
   1:  PR[91,1] = PR[90,1] + 16.034;
   1:  PR[91,2] = PR[90,2] + -16.968;
   1:L PR[91] R[100]mm/sec CNT100;
   1:  PR[91,1] = PR[90,1] + 19.725;
   1:  PR[91,2] = PR[90,2] + -18.490;
   1:L PR[91] R[100]mm/sec CNT100;
   1:  PR[91,1] = PR[90,1] + 20.251;
   1:  PR[91,2] = PR[90,2] + -18.631;
   1:L PR[91] R[100]mm/sec CNT100;
   1:  PR[91,1] = PR[90,1] + 24.153;
   1:  PR[91,2] = PR[90,2] + -19.139;
   1:L PR[91] R[100]mm/sec CNT100;
   1:  PR[91,1] = PR[90,1] + 24.768;
   1:  PR[91,2] = PR[90,2] + -19.192;
   1:L PR[91] R[100]mm/sec CNT100;
   1:  PR[91,1] = PR[90,1] + 25.380;
   1:  PR[91,2] = PR[90,2] + -19.139;
   1:L PR[91] R[100]mm/sec CNT100;
   1:  PR[91,1] = PR[90,1] + 29.249;
   1:  PR[91,2] = PR[90,2] + -18.622;
   1:L PR[91] R[100]mm/sec CNT100;
   1:  PR[91,1] = PR[90,1] + 29.789;
   1:  PR[91,2] = PR[90,2] + -18.477;
   1:L PR[91] R[100]mm/sec CNT100;
   1:  PR[91,1] = PR[90,1] + 30.450;
   1:  PR[91,2] = PR[90,2] + -18.169;
   1:L PR[91] R[100]mm/sec CNT100;
   1:  PR[91,1] = PR[90,1] + 34.024;
   1:  PR[91,2] = PR[90,2] + -16.681;
   1:L PR[91] R[100]mm/sec CNT100;
   1:  PR[91,1] = PR[90,1] + 34.539;
   1:  PR[91,2] = PR[90,2] + -16.320;
   1:L PR[91] R[100]mm/sec CNT100;
   1:  PR[91,1] = PR[90,1] + 37.568;
   1:  PR[91,2] = PR[90,2] + -13.991;
   1:L PR[91] R[100]mm/sec CNT100;
   1:  PR[91,1] = PR[90,1] + 38.026;
   1:  PR[91,2] = PR[90,2] + -13.533;
   1:L PR[91] R[100]mm/sec CNT100;
   1:  PR[91,1] = PR[90,1] + 40.324;
   1:  PR[91,2] = PR[90,2] + -10.530;
   1:L PR[91] R[100]mm/sec CNT100;
   1:  PR[91,1] = PR[90,1] + 40.733;
   1:  PR[91,2] = PR[90,2] + -9.947;
   1:L PR[91] R[100]mm/sec CNT100;
   1:  PR[91,1] = PR[90,1] + 41.032;
   1:  PR[91,2] = PR[90,2] + -9.305;
   1:L PR[91] R[100]mm/sec CNT100;
   1:  PR[91,1] = PR[90,1] + 42.471;
   1:  PR[91,2] = PR[90,2] + -5.824;
   1:L PR[91] R[100]mm/sec CNT100;
   1:  PR[91,1] = PR[90,1] + 42.635;
   1:  PR[91,2] = PR[90,2] + -5.212;
   1:L PR[91] R[100]mm/sec CNT100;
   1:  PR[91,1] = PR[90,1] + 42.704;
   1:  PR[91,2] = PR[90,2] + -4.424;
   1:L PR[91] R[100]mm/sec CNT100;
   1:  PR[91,1] = PR[90,1] + 43.146;
   1:  PR[91,2] = PR[90,2] + -0.638;
   1:L PR[91] R[100]mm/sec CNT100;
   1:  PR[91,1] = PR[90,1] + 43.128;
   1:  PR[91,2] = PR[90,2] + 0.046;
   1:L PR[91] R[100]mm/sec CNT100;
   1:  PR[91,1] = PR[90,1] + 42.647;
   1:  PR[91,2] = PR[90,2] + 3.711;
   1:L PR[91] R[100]mm/sec CNT100;
   1:  PR[91,1] = PR[90,1] + 42.471;
   1:  PR[91,2] = PR[90,2] + 4.366;
   1:L PR[91] R[100]mm/sec CNT100;
   1:  PR[91,1] = PR[90,1] + 41.032;
   1:  PR[91,2] = PR[90,2] + 7.846;
   1:L PR[91] R[100]mm/sec CNT100;
   1:  PR[91,1] = PR[90,1] + 40.733;
   1:  PR[91,2] = PR[90,2] + 8.488;
   1:L PR[91] R[100]mm/sec CNT100;
   1:  PR[91,1] = PR[90,1] + 40.324;
   1:  PR[91,2] = PR[90,2] + 9.072;
   1:L PR[91] R[100]mm/sec CNT100;
   1:  PR[91,1] = PR[90,1] + 38.025;
   1:  PR[91,2] = PR[90,2] + 12.075;
   1:L PR[91] R[100]mm/sec CNT100;
   1:  PR[91,1] = PR[90,1] + 37.567;
   1:  PR[91,2] = PR[90,2] + 12.533;
   1:L PR[91] R[100]mm/sec CNT100;
   1:  PR[91,1] = PR[90,1] + 34.538;
   1:  PR[91,2] = PR[90,2] + 14.862;
   1:L PR[91] R[100]mm/sec CNT100;
   1:  PR[91,1] = PR[90,1] + 33.989;
   1:  PR[91,2] = PR[90,2] + 15.247;
   1:L PR[91] R[100]mm/sec CNT100;
   1:  PR[91,1] = PR[90,1] + 33.379;
   1:  PR[91,2] = PR[90,2] + 15.531;
   1:L PR[91] R[100]mm/sec CNT100;
   1:  PR[91,1] = PR[90,1] + 29.828;
   1:  PR[91,2] = PR[90,2] + 17.008;
   1:L PR[91] R[100]mm/sec CNT100;
   1:  PR[91,1] = PR[90,1] + 29.246;
   1:  PR[91,2] = PR[90,2] + 17.164;
   1:L PR[91] R[100]mm/sec CNT100;
   1:  PR[91,1] = PR[90,1] + 25.377;
   1:  PR[91,2] = PR[90,2] + 17.680;
   1:L PR[91] R[100]mm/sec CNT100;
   1:  PR[91,1] = PR[90,1] + 24.766;
   1:  PR[91,2] = PR[90,2] + 17.734;
   1:L PR[91] R[100]mm/sec CNT100;
   1:  PR[91,1] = PR[90,1] + 24.150;
   1:  PR[91,2] = PR[90,2] + 17.680;
   1:L PR[91] R[100]mm/sec CNT100;
   1:  PR[91,1] = PR[90,1] + 20.249;
   1:  PR[91,2] = PR[90,2] + 17.172;
   1:L PR[91] R[100]mm/sec CNT100;
   1:  PR[91,1] = PR[90,1] + 19.767;
   1:  PR[91,2] = PR[90,2] + 17.043;
   1:L PR[91] R[100]mm/sec CNT100;
   1:  PR[91,1] = PR[90,1] + 19.155;
   1:  PR[91,2] = PR[90,2] + 16.757;
   1:L PR[91] R[100]mm/sec CNT100;
   1:  PR[91,1] = PR[90,1] + 15.490;
   1:  PR[91,2] = PR[90,2] + 15.247;
   1:L PR[91] R[100]mm/sec CNT100;
   1:  PR[91,1] = PR[90,1] + 15.067;
   1:  PR[91,2] = PR[90,2] + 14.951;
   1:L PR[91] R[100]mm/sec CNT100;
   1:  PR[91,1] = PR[90,1] + 11.873;
   1:  PR[91,2] = PR[90,2] + 12.508;
   1:L PR[91] R[100]mm/sec CNT100;
   1:  PR[91,1] = PR[90,1] + 11.527;
   1:  PR[91,2] = PR[90,2] + 12.162;
   1:L PR[91] R[100]mm/sec CNT100;
   1:  PR[91,1] = PR[90,1] + 9.049;
   1:  PR[91,2] = PR[90,2] + 8.939;
   1:L PR[91] R[100]mm/sec CNT100;
   1:  PR[91,1] = PR[90,1] + 8.753;
   1:  PR[91,2] = PR[90,2] + 8.515;
   1:L PR[91] R[100]mm/sec CNT100;
   1:  PR[91,1] = PR[90,1] + 8.534;
   1:  PR[91,2] = PR[90,2] + 8.047;
   1:L PR[91] R[100]mm/sec CNT100;
   1:  PR[91,1] = PR[90,1] + 6.970;
   1:  PR[91,2] = PR[90,2] + 4.277;
   1:L PR[91] R[100]mm/sec CNT100;
   1:  PR[91,1] = PR[90,1] + 6.862;
   1:  PR[91,2] = PR[90,2] + 3.874;
   1:L PR[91] R[100]mm/sec CNT100;
   1:  PR[91,1] = PR[90,1] + 6.811;
   1:  PR[91,2] = PR[90,2] + 3.287;
   1:L PR[91] R[100]mm/sec CNT100;
   1:  PR[91,1] = PR[90,1] + 6.282;
   1:  PR[91,2] = PR[90,2] + -0.772;
   1:L PR[91] R[100]mm/sec CNT100;
   1:  PR[91,1] = PR[90,1] + 6.336;
   1:  PR[91,2] = PR[90,2] + -1.394;
   1:L PR[91] R[100]mm/sec CNT100;
   1:  PR[91,1] = PR[90,1] + 6.851;
   1:  PR[91,2] = PR[90,2] + -5.290;
   1:L PR[91] R[100]mm/sec CNT100;
   1:  PR[91,1] = PR[90,1] + 6.970;
   1:  PR[91,2] = PR[90,2] + -5.736;
   1:L PR[91] R[100]mm/sec CNT100;
   1:  PR[91,1] = PR[90,1] + 8.535;
   1:  PR[91,2] = PR[90,2] + -9.506;
   1:L PR[91] R[100]mm/sec CNT100;
   1:  PR[91,1] = PR[90,1] + 8.753;
   1:  PR[91,2] = PR[90,2] + -9.975;
   1:L PR[91] R[100]mm/sec CNT100;
   1:  PR[91,1] = PR[90,1] + 9.050;
   1:  PR[91,2] = PR[90,2] + -10.398;
   1:L PR[91] R[100]mm/sec CNT100;
   1:  PR[91,1] = PR[90,1] + 11.528;
   1:  PR[91,2] = PR[90,2] + -13.622;
   1:L PR[91] R[100]mm/sec CNT100;
   1:  PR[91,1] = PR[90,1] + 11.874;
   1:  PR[91,2] = PR[90,2] + -13.968;
   1:L PR[91] R[100]mm/sec CNT100TB   .50sec,CALL END_PUD;
   1:  PR[92] = PR[91];
   1:  PR[92,3] = PR[92,3] + 20;
   1:J PR[92] 10% FINE;
   1:  PR[91,1] = PR[90,1] + 59.086;
   1:  PR[91,2] = PR[90,2] + -12.393;
   1:  PR[92] = PR[91];
   1:  PR[92,3] = PR[92,3] + 20;
   1:J PR[92] 10% FINE;
   1:L PR[91] R[100]mm/sec CNT100;
   1:  CALL LASER_DRAHT_START;
   1:  PR[91,1] = PR[90,1] + 60.293;
   1:  PR[91,2] = PR[90,2] + -13.557;
   1:L PR[91] R[100]mm/sec CNT100;
   1:  PR[91,1] = PR[90,1] + 62.143;
   1:  PR[91,2] = PR[90,2] + -15.300;
   1:L PR[91] R[100]mm/sec CNT100;
   1:  PR[91,1] = PR[90,1] + 63.971;
   1:  PR[91,2] = PR[90,2] + -16.401;
   1:L PR[91] R[100]mm/sec CNT100;
   1:  PR[91,1] = PR[90,1] + 65.772;
   1:  PR[91,2] = PR[90,2] + -17.456;
   1:L PR[91] R[100]mm/sec CNT100;
   1:  PR[91,1] = PR[90,1] + 68.248;
   1:  PR[91,2] = PR[90,2] + -18.274;
   1:L PR[91] R[100]mm/sec CNT100;
   1:  PR[91,1] = PR[90,1] + 69.782;
   1:  PR[91,2] = PR[90,2] + -18.759;
   1:L PR[91] R[100]mm/sec CNT100;
   1:  PR[91,1] = PR[90,1] + 72.825;
   1:  PR[91,2] = PR[90,2] + -19.060;
   1:L PR[91] R[100]mm/sec CNT100;
   1:  PR[91,1] = PR[90,1] + 73.969;
   1:  PR[91,2] = PR[90,2] + -19.158;
   1:L PR[91] R[100]mm/sec CNT100;
   1:  PR[91,1] = PR[90,1] + 78.141;
   1:  PR[91,2] = PR[90,2] + -18.634;
   1:L PR[91] R[100]mm/sec CNT100;
   1:  PR[91,1] = PR[90,1] + 81.686;
   1:  PR[91,2] = PR[90,2] + -17.372;
   1:L PR[91] R[100]mm/sec CNT100;
   1:  PR[91,1] = PR[90,1] + 82.061;
   1:  PR[91,2] = PR[90,2] + -17.234;
   1:L PR[91] R[100]mm/sec CNT100;
   1:  PR[91,1] = PR[90,1] + 85.575;
   1:  PR[91,2] = PR[90,2] + -15.011;
   1:L PR[91] R[100]mm/sec CNT100;
   1:  PR[91,1] = PR[90,1] + 88.491;
   1:  PR[91,2] = PR[90,2] + -12.096;
   1:L PR[91] R[100]mm/sec CNT100;
   1:  PR[91,1] = PR[90,1] + 90.677;
   1:  PR[91,2] = PR[90,2] + -8.631;
   1:L PR[91] R[100]mm/sec CNT100;
   1:  PR[91,1] = PR[90,1] + 92.020;
   1:  PR[91,2] = PR[90,2] + -4.770;
   1:L PR[91] R[100]mm/sec CNT100;
   1:  PR[91,1] = PR[90,1] + 92.467;
   1:  PR[91,2] = PR[90,2] + -0.729;
   1:L PR[91] R[100]mm/sec CNT100;
   1:  PR[91,1] = PR[90,1] + 92.020;
   1:  PR[91,2] = PR[90,2] + 3.311;
   1:L PR[91] R[100]mm/sec CNT100;
   1:  PR[91,1] = PR[90,1] + 90.677;
   1:  PR[91,2] = PR[90,2] + 7.172;
   1:L PR[91] R[100]mm/sec CNT100;
   1:  PR[91,1] = PR[90,1] + 88.491;
   1:  PR[91,2] = PR[90,2] + 10.637;
   1:L PR[91] R[100]mm/sec CNT100;
   1:  PR[91,1] = PR[90,1] + 85.575;
   1:  PR[91,2] = PR[90,2] + 13.552;
   1:L PR[91] R[100]mm/sec CNT100;
   1:  PR[91,1] = PR[90,1] + 82.069;
   1:  PR[91,2] = PR[90,2] + 15.770;
   1:L PR[91] R[100]mm/sec CNT100;
   1:  PR[91,1] = PR[90,1] + 78.143;
   1:  PR[91,2] = PR[90,2] + 17.175;
   1:L PR[91] R[100]mm/sec CNT100;
   1:  PR[91,1] = PR[90,1] + 74.809;
   1:  PR[91,2] = PR[90,2] + 17.581;
   1:L PR[91] R[100]mm/sec CNT100;
   1:  PR[91,1] = PR[90,1] + 73.972;
   1:  PR[91,2] = PR[90,2] + 17.696;
   1:L PR[91] R[100]mm/sec CNT100;
   1:  PR[91,1] = PR[90,1] + 70.968;
   1:  PR[91,2] = PR[90,2] + 17.396;
   1:L PR[91] R[100]mm/sec CNT100;
   1:  PR[91,1] = PR[90,1] + 69.783;
   1:  PR[91,2] = PR[90,2] + 17.297;
   1:L PR[91] R[100]mm/sec CNT100;
   1:  PR[91,1] = PR[90,1] + 67.265;
   1:  PR[91,2] = PR[90,2] + 16.462;
   1:L PR[91] R[100]mm/sec CNT100;
   1:  PR[91,1] = PR[90,1] + 65.772;
   1:  PR[91,2] = PR[90,2] + 15.993;
   1:L PR[91] R[100]mm/sec CNT100;
   1:  PR[91,1] = PR[90,1] + 63.838;
   1:  PR[91,2] = PR[90,2] + 14.826;
   1:L PR[91] R[100]mm/sec CNT100;
   1:  PR[91,1] = PR[90,1] + 62.143;
   1:  PR[91,2] = PR[90,2] + 13.837;
   1:L PR[91] R[100]mm/sec CNT100;
   1:  PR[91,1] = PR[90,1] + 60.804;
   1:  PR[91,2] = PR[90,2] + 12.545;
   1:L PR[91] R[100]mm/sec CNT100;
   1:  PR[91,1] = PR[90,1] + 59.084;
   1:  PR[91,2] = PR[90,2] + 10.928;
   1:L PR[91] R[100]mm/sec CNT100;
   1:  PR[91,1] = PR[90,1] + 58.273;
   1:  PR[91,2] = PR[90,2] + 9.680;
   1:L PR[91] R[100]mm/sec CNT100;
   1:  PR[91,1] = PR[90,1] + 56.759;
   1:  PR[91,2] = PR[90,2] + 7.403;
   1:L PR[91] R[100]mm/sec CNT100;
   1:  PR[91,1] = PR[90,1] + 55.312;
   1:  PR[91,2] = PR[90,2] + 3.452;
   1:L PR[91] R[100]mm/sec CNT100;
   1:  PR[91,1] = PR[90,1] + 55.212;
   1:  PR[91,2] = PR[90,2] + 2.599;
   1:L PR[91] R[100]mm/sec CNT100;
   1:  PR[91,1] = PR[90,1] + 55.211;
   1:  PR[91,2] = PR[90,2] + 2.366;
   1:L PR[91] R[100]mm/sec CNT100;
   1:  PR[91,1] = PR[90,1] + 54.847;
   1:  PR[91,2] = PR[90,2] + -0.750;
   1:L PR[91] R[100]mm/sec CNT100;
   1:  PR[91,1] = PR[90,1] + 54.928;
   1:  PR[91,2] = PR[90,2] + -1.594;
   1:L PR[91] R[100]mm/sec CNT100;
   1:  PR[91,1] = PR[90,1] + 55.312;
   1:  PR[91,2] = PR[90,2] + -4.913;
   1:L PR[91] R[100]mm/sec CNT100;
   1:  PR[91,1] = PR[90,1] + 56.761;
   1:  PR[91,2] = PR[90,2] + -8.866;
   1:L PR[91] R[100]mm/sec CNT100;
   1:  PR[91,1] = PR[90,1] + 59.086;
   1:  PR[91,2] = PR[90,2] + -12.393;
   1:L PR[91] R[100]mm/sec CNT100TB   .50sec,CALL END_PUD;
   1:  PR[92] = PR[91];
   1:  PR[92,3] = PR[92,3] + 20;
   1:J PR[92] 10% FINE;
   1:  PR[91,1] = PR[90,1] + -40.837;
   1:  PR[91,2] = PR[90,2] + 7.347;
   1:  PR[92] = PR[91];
   1:  PR[92,3] = PR[92,3] + 20;
   1:J PR[92] 10% FINE;
   1:L PR[91] R[100]mm/sec CNT100;
   1:  CALL LASER_DRAHT_START;
   1:  PR[91,1] = PR[90,1] + -41.039;
   1:  PR[91,2] = PR[90,2] + 6.912;
   1:L PR[91] R[100]mm/sec CNT100;
   1:  PR[91,1] = PR[90,1] + -42.167;
   1:  PR[91,2] = PR[90,2] + 3.679;
   1:L PR[91] R[100]mm/sec CNT100;
   1:  PR[91,1] = PR[90,1] + -42.292;
   1:  PR[91,2] = PR[90,2] + 3.211;
   1:L PR[91] R[100]mm/sec CNT100;
   1:  PR[91,1] = PR[90,1] + -42.343;
   1:  PR[91,2] = PR[90,2] + 2.632;
   1:L PR[91] R[100]mm/sec CNT100;
   1:  PR[91,1] = PR[90,1] + -42.723;
   1:  PR[91,2] = PR[90,2] + -0.754;
   1:L PR[91] R[100]mm/sec CNT100;
   1:  PR[91,1] = PR[90,1] + -42.678;
   1:  PR[91,2] = PR[90,2] + -1.274;
   1:L PR[91] R[100]mm/sec CNT100;
   1:  PR[91,1] = PR[90,1] + -42.298;
   1:  PR[91,2] = PR[90,2] + -4.646;
   1:L PR[91] R[100]mm/sec CNT100;
   1:  PR[91,1] = PR[90,1] + -42.167;
   1:  PR[91,2] = PR[90,2] + -5.137;
   1:L PR[91] R[100]mm/sec CNT100;
   1:  PR[91,1] = PR[90,1] + -41.039;
   1:  PR[91,2] = PR[90,2] + -8.371;
   1:L PR[91] R[100]mm/sec CNT100;
   1:  PR[91,1] = PR[90,1] + -40.837;
   1:  PR[91,2] = PR[90,2] + -8.806;
   1:L PR[91] R[100]mm/sec CNT100;
   1:  PR[91,1] = PR[90,1] + -38.985;
   1:  PR[91,2] = PR[90,2] + -11.762;
   1:L PR[91] R[100]mm/sec CNT100;
   1:  PR[91,1] = PR[90,1] + -38.737;
   1:  PR[91,2] = PR[90,2] + -12.115;
   1:L PR[91] R[100]mm/sec CNT100;
   1:  PR[91,1] = PR[90,1] + -35.914;
   1:  PR[91,2] = PR[90,2] + -14.949;
   1:L PR[91] R[100]mm/sec CNT100;
   1:  PR[91,1] = PR[90,1] + -35.616;
   1:  PR[91,2] = PR[90,2] + -15.158;
   1:L PR[91] R[100]mm/sec CNT100;
   1:  PR[91,1] = PR[90,1] + -32.543;
   1:  PR[91,2] = PR[90,2] + -17.099;
   1:L PR[91] R[100]mm/sec CNT100;
   1:  PR[91,1] = PR[90,1] + -32.290;
   1:  PR[91,2] = PR[90,2] + -17.218;
   1:L PR[91] R[100]mm/sec CNT100;
   1:  PR[91,1] = PR[90,1] + -28.724;
   1:  PR[91,2] = PR[90,2] + -18.475;
   1:L PR[91] R[100]mm/sec CNT100;
   1:  PR[91,1] = PR[90,1] + -28.577;
   1:  PR[91,2] = PR[90,2] + -18.514;
   1:L PR[91] R[100]mm/sec CNT100;
   1:  PR[91,1] = PR[90,1] + -28.319;
   1:  PR[91,2] = PR[90,2] + -18.537;
   1:L PR[91] R[100]mm/sec CNT100;
   1:  PR[91,1] = PR[90,1] + -24.525;
   1:  PR[91,2] = PR[90,2] + -18.980;
   1:L PR[91] R[100]mm/sec CNT100;
   1:  PR[91,1] = PR[90,1] + -20.455;
   1:  PR[91,2] = PR[90,2] + -18.540;
   1:L PR[91] R[100]mm/sec CNT100;
   1:  PR[91,1] = PR[90,1] + -16.577;
   1:  PR[91,2] = PR[90,2] + -17.192;
   1:L PR[91] R[100]mm/sec CNT100;
   1:  PR[91,1] = PR[90,1] + -15.160;
   1:  PR[91,2] = PR[90,2] + -16.307;
   1:L PR[91] R[100]mm/sec CNT100;
   1:  PR[91,1] = PR[90,1] + -13.076;
   1:  PR[91,2] = PR[90,2] + -15.031;
   1:L PR[91] R[100]mm/sec CNT100;
   1:  PR[91,1] = PR[90,1] + -10.125;
   1:  PR[91,2] = PR[90,2] + -12.150;
   1:L PR[91] R[100]mm/sec CNT100;
   1:  PR[91,1] = PR[90,1] + -7.899;
   1:  PR[91,2] = PR[90,2] + -8.685;
   1:L PR[91] R[100]mm/sec CNT100;
   1:  PR[91,1] = PR[90,1] + -6.516;
   1:  PR[91,2] = PR[90,2] + -4.813;
   1:L PR[91] R[100]mm/sec CNT100;
   1:  PR[91,1] = PR[90,1] + -6.050;
   1:  PR[91,2] = PR[90,2] + -0.729;
   1:L PR[91] R[100]mm/sec CNT100;
   1:  PR[91,1] = PR[90,1] + -6.492;
   1:  PR[91,2] = PR[90,2] + 3.146;
   1:L PR[91] R[100]mm/sec CNT100;
   1:  PR[91,1] = PR[90,1] + -6.516;
   1:  PR[91,2] = PR[90,2] + 3.353;
   1:L PR[91] R[100]mm/sec CNT100;
   1:  PR[91,1] = PR[90,1] + -7.899;
   1:  PR[91,2] = PR[90,2] + 7.226;
   1:L PR[91] R[100]mm/sec CNT100;
   1:  PR[91,1] = PR[90,1] + -10.125;
   1:  PR[91,2] = PR[90,2] + 10.691;
   1:L PR[91] R[100]mm/sec CNT100;
   1:  PR[91,1] = PR[90,1] + -13.076;
   1:  PR[91,2] = PR[90,2] + 13.573;
   1:L PR[91] R[100]mm/sec CNT100;
   1:  PR[91,1] = PR[90,1] + -15.160;
   1:  PR[91,2] = PR[90,2] + 14.848;
   1:L PR[91] R[100]mm/sec CNT100;
   1:  PR[91,1] = PR[90,1] + -16.577;
   1:  PR[91,2] = PR[90,2] + 15.733;
   1:L PR[91] R[100]mm/sec CNT100;
   1:  PR[91,1] = PR[90,1] + -20.455;
   1:  PR[91,2] = PR[90,2] + 17.081;
   1:L PR[91] R[100]mm/sec CNT100;
   1:  PR[91,1] = PR[90,1] + -24.527;
   1:  PR[91,2] = PR[90,2] + 17.522;
   1:L PR[91] R[100]mm/sec CNT100;
   1:  PR[91,1] = PR[90,1] + -28.551;
   1:  PR[91,2] = PR[90,2] + 17.062;
   1:L PR[91] R[100]mm/sec CNT100;
   1:  PR[91,1] = PR[90,1] + -28.724;
   1:  PR[91,2] = PR[90,2] + 17.016;
   1:L PR[91] R[100]mm/sec CNT100;
   1:  PR[91,1] = PR[90,1] + -32.290;
   1:  PR[91,2] = PR[90,2] + 15.759;
   1:L PR[91] R[100]mm/sec CNT100;
   1:  PR[91,1] = PR[90,1] + -32.543;
   1:  PR[91,2] = PR[90,2] + 15.640;
   1:L PR[91] R[100]mm/sec CNT100;
   1:  PR[91,1] = PR[90,1] + -35.616;
   1:  PR[91,2] = PR[90,2] + 13.699;
   1:L PR[91] R[100]mm/sec CNT100;
   1:  PR[91,1] = PR[90,1] + -35.914;
   1:  PR[91,2] = PR[90,2] + 13.490;
   1:L PR[91] R[100]mm/sec CNT100;
   1:  PR[91,1] = PR[90,1] + -38.737;
   1:  PR[91,2] = PR[90,2] + 10.656;
   1:L PR[91] R[100]mm/sec CNT100;
   1:  PR[91,1] = PR[90,1] + -38.984;
   1:  PR[91,2] = PR[90,2] + 10.303;
   1:L PR[91] R[100]mm/sec CNT100;
   1:  PR[91,1] = PR[90,1] + -40.837;
   1:  PR[91,2] = PR[90,2] + 7.347;
   1:L PR[91] R[100]mm/sec CNT100TB   .50sec,CALL END_PUD;
   1:  PR[92] = PR[91];
   1:  PR[92,3] = PR[92,3] + 20;
   1:J PR[92] 10% FINE;
   1:  PR[91,1] = PR[90,1] + -83.415;
   1:  PR[91,2] = PR[90,2] + 14.998;
   1:  PR[92] = PR[91];
   1:  PR[92,3] = PR[92,3] + 20;
   1:J PR[92] 10% FINE;
   1:L PR[91] R[100]mm/sec CNT100;
   1:  CALL LASER_DRAHT_START;
   1:  PR[91,1] = PR[90,1] + -86.519;
   1:  PR[91,2] = PR[90,2] + 12.750;
   1:L PR[91] R[100]mm/sec CNT100;
   1:  PR[91,1] = PR[90,1] + -89.079;
   1:  PR[91,2] = PR[90,2] + 9.920;
   1:L PR[91] R[100]mm/sec CNT100;
   1:  PR[91,1] = PR[90,1] + -90.989;
   1:  PR[91,2] = PR[90,2] + 6.634;
   1:L PR[91] R[100]mm/sec CNT100;
   1:  PR[91,1] = PR[90,1] + -92.167;
   1:  PR[91,2] = PR[90,2] + 3.033;
   1:L PR[91] R[100]mm/sec CNT100;
   1:  PR[91,1] = PR[90,1] + -92.552;
   1:  PR[91,2] = PR[90,2] + -0.594;
   1:L PR[91] R[100]mm/sec CNT100;
   1:  PR[91,1] = PR[90,1] + -92.516;
   1:  PR[91,2] = PR[90,2] + -0.742;
   1:L PR[91] R[100]mm/sec CNT100;
   1:  PR[91,1] = PR[90,1] + -92.124;
   1:  PR[91,2] = PR[90,2] + -4.484;
   1:L PR[91] R[100]mm/sec CNT100;
   1:  PR[91,1] = PR[90,1] + -92.092;
   1:  PR[91,2] = PR[90,2] + -4.604;
   1:L PR[91] R[100]mm/sec CNT100;
   1:  PR[91,1] = PR[90,1] + -90.966;
   1:  PR[91,2] = PR[90,2] + -8.078;
   1:L PR[91] R[100]mm/sec CNT100;
   1:  PR[91,1] = PR[90,1] + -90.932;
   1:  PR[91,2] = PR[90,2] + -8.151;
   1:L PR[91] R[100]mm/sec CNT100;
   1:  PR[91,1] = PR[90,1] + -89.070;
   1:  PR[91,2] = PR[90,2] + -11.382;
   1:L PR[91] R[100]mm/sec CNT100;
   1:  PR[91,1] = PR[90,1] + -89.064;
   1:  PR[91,2] = PR[90,2] + -11.391;
   1:L PR[91] R[100]mm/sec CNT100;
   1:  PR[91,1] = PR[90,1] + -86.510;
   1:  PR[91,2] = PR[90,2] + -14.226;
   1:L PR[91] R[100]mm/sec CNT100;
   1:  PR[91,1] = PR[90,1] + -83.462;
   1:  PR[91,2] = PR[90,2] + -16.448;
   1:L PR[91] R[100]mm/sec CNT100;
   1:  PR[91,1] = PR[90,1] + -79.943;
   1:  PR[91,2] = PR[90,2] + -18.018;
   1:L PR[91] R[100]mm/sec CNT100;
   1:  PR[91,1] = PR[90,1] + -76.158;
   1:  PR[91,2] = PR[90,2] + -18.839;
   1:L PR[91] R[100]mm/sec CNT100;
   1:  PR[91,1] = PR[90,1] + -72.275;
   1:  PR[91,2] = PR[90,2] + -18.873;
   1:L PR[91] R[100]mm/sec CNT100;
   1:  PR[91,1] = PR[90,1] + -68.461;
   1:  PR[91,2] = PR[90,2] + -18.113;
   1:L PR[91] R[100]mm/sec CNT100;
   1:  PR[91,1] = PR[90,1] + -64.885;
   1:  PR[91,2] = PR[90,2] + -16.588;
   1:L PR[91] R[100]mm/sec CNT100;
   1:  PR[91,1] = PR[90,1] + -61.704;
   1:  PR[91,2] = PR[90,2] + -14.363;
   1:L PR[91] R[100]mm/sec CNT100;
   1:  PR[91,1] = PR[90,1] + -59.064;
   1:  PR[91,2] = PR[90,2] + -11.529;
   1:L PR[91] R[100]mm/sec CNT100;
   1:  PR[91,1] = PR[90,1] + -57.083;
   1:  PR[91,2] = PR[90,2] + -8.212;
   1:L PR[91] R[100]mm/sec CNT100;
   1:  PR[91,1] = PR[90,1] + -55.857;
   1:  PR[91,2] = PR[90,2] + -4.558;
   1:L PR[91] R[100]mm/sec CNT100;
   1:  PR[91,1] = PR[90,1] + -55.668;
   1:  PR[91,2] = PR[90,2] + -2.815;
   1:L PR[91] R[100]mm/sec CNT100;
   1:  PR[91,1] = PR[90,1] + -55.618;
   1:  PR[91,2] = PR[90,2] + -1.089;
   1:L PR[91] R[100]mm/sec CNT100;
   1:  PR[91,1] = PR[90,1] + -55.578;
   1:  PR[91,2] = PR[90,2] + -0.668;
   1:L PR[91] R[100]mm/sec CNT100;
   1:  PR[91,1] = PR[90,1] + -55.613;
   1:  PR[91,2] = PR[90,2] + 0.420;
   1:L PR[91] R[100]mm/sec CNT100;
   1:  PR[91,1] = PR[90,1] + -55.902;
   1:  PR[91,2] = PR[90,2] + 3.098;
   1:L PR[91] R[100]mm/sec CNT100;
   1:  PR[91,1] = PR[90,1] + -57.123;
   1:  PR[91,2] = PR[90,2] + 6.752;
   1:L PR[91] R[100]mm/sec CNT100;
   1:  PR[91,1] = PR[90,1] + -59.096;
   1:  PR[91,2] = PR[90,2] + 10.069;
   1:L PR[91] R[100]mm/sec CNT100;
   1:  PR[91,1] = PR[90,1] + -61.725;
   1:  PR[91,2] = PR[90,2] + 12.904;
   1:L PR[91] R[100]mm/sec CNT100;
   1:  PR[91,1] = PR[90,1] + -64.896;
   1:  PR[91,2] = PR[90,2] + 15.132;
   1:L PR[91] R[100]mm/sec CNT100;
   1:  PR[91,1] = PR[90,1] + -67.021;
   1:  PR[91,2] = PR[90,2] + 16.050;
   1:L PR[91] R[100]mm/sec CNT100;
   1:  PR[91,1] = PR[90,1] + -68.452;
   1:  PR[91,2] = PR[90,2] + 16.656;
   1:L PR[91] R[100]mm/sec CNT100;
   1:  PR[91,1] = PR[90,1] + -72.257;
   1:  PR[91,2] = PR[90,2] + 17.419;
   1:L PR[91] R[100]mm/sec CNT100;
   1:  PR[91,1] = PR[90,1] + -76.127;
   1:  PR[91,2] = PR[90,2] + 17.388;
   1:L PR[91] R[100]mm/sec CNT100;
   1:  PR[91,1] = PR[90,1] + -79.901;
   1:  PR[91,2] = PR[90,2] + 16.568;
   1:L PR[91] R[100]mm/sec CNT100;
   1:  PR[91,1] = PR[90,1] + -83.415;
   1:  PR[91,2] = PR[90,2] + 14.998;
   1:L PR[91] R[100]mm/sec CNT100TB   .50sec,CALL END_PUD;
   1:  PR[92] = PR[91];
   1:  PR[92,3] = PR[92,3] + 20;
   1:J PR[92] 10% FINE;
   1:  PR[91] = PR[90];
   1:  PR[91,1] = PR[90,1] + 80.831;
   1:  PR[91,2] = PR[90,2] + -17.694;
   1:  PR[91,3] = PR[90,3] + 20.995;
   1:  PR[92] = PR[91];
   1:  PR[92,3] = PR[92,3] + 20;
   1:J PR[92] 10% FINE;
   1:L PR[91] R[100]mm/sec CNT100;
   1:  CALL LASER_DRAHT_START;
   1:  PR[91,1] = PR[90,1] + 81.864;
   1:  PR[91,2] = PR[90,2] + -17.313;
   1:L PR[91] R[100]mm/sec CNT100;
   1:  PR[91,1] = PR[90,1] + 85.391;
   1:  PR[91,2] = PR[90,2] + -15.076;
   1:L PR[91] R[100]mm/sec CNT100;
   1:  PR[91,1] = PR[90,1] + 88.316;
   1:  PR[91,2] = PR[90,2] + -12.145;
   1:L PR[91] R[100]mm/sec CNT100;
   1:  PR[91,1] = PR[90,1] + 90.510;
   1:  PR[91,2] = PR[90,2] + -8.661;
   1:L PR[91] R[100]mm/sec CNT100;
   1:  PR[91,1] = PR[90,1] + 91.869;
   1:  PR[91,2] = PR[90,2] + -4.791;
   1:L PR[91] R[100]mm/sec CNT100;
   1:  PR[91,1] = PR[90,1] + 92.323;
   1:  PR[91,2] = PR[90,2] + -0.849;
   1:L PR[91] R[100]mm/sec CNT100;
   1:  PR[91,1] = PR[90,1] + 92.347;
   1:  PR[91,2] = PR[90,2] + -0.692;
   1:L PR[91] R[100]mm/sec CNT100;
   1:  PR[91,1] = PR[90,1] + 91.953;
   1:  PR[91,2] = PR[90,2] + 2.747;
   1:L PR[91] R[100]mm/sec CNT100;
   1:  PR[91,1] = PR[90,1] + 91.901;
   1:  PR[91,2] = PR[90,2] + 3.027;
   1:L PR[91] R[100]mm/sec CNT100;
   1:  PR[91,1] = PR[90,1] + 91.867;
   1:  PR[91,2] = PR[90,2] + 3.336;
   1:L PR[91] R[100]mm/sec CNT100;
   1:  PR[91,1] = PR[90,1] + 90.510;
   1:  PR[91,2] = PR[90,2] + 7.202;
   1:L PR[91] R[100]mm/sec CNT100;
   1:  PR[91,1] = PR[90,1] + 88.316;
   1:  PR[91,2] = PR[90,2] + 10.686;
   1:L PR[91] R[100]mm/sec CNT100;
   1:  PR[91,1] = PR[90,1] + 85.391;
   1:  PR[91,2] = PR[90,2] + 13.617;
   1:L PR[91] R[100]mm/sec CNT100;
   1:  PR[91,1] = PR[90,1] + 81.874;
   1:  PR[91,2] = PR[90,2] + 15.848;
   1:L PR[91] R[100]mm/sec CNT100;
   1:  PR[91,1] = PR[90,1] + 78.992;
   1:  PR[91,2] = PR[90,2] + 16.872;
   1:L PR[91] R[100]mm/sec CNT100;
   1:  PR[91,1] = PR[90,1] + 77.920;
   1:  PR[91,2] = PR[90,2] + 17.269;
   1:L PR[91] R[100]mm/sec CNT100;
   1:  PR[91,1] = PR[90,1] + 75.202;
   1:  PR[91,2] = PR[90,2] + 17.601;
   1:L PR[91] R[100]mm/sec CNT100;
   1:  PR[91,1] = PR[90,1] + 73.738;
   1:  PR[91,2] = PR[90,2] + 17.801;
   1:L PR[91] R[100]mm/sec CNT100;
   1:  PR[91,1] = PR[90,1] + 71.378;
   1:  PR[91,2] = PR[90,2] + 17.566;
   1:L PR[91] R[100]mm/sec CNT100;
   1:  PR[91,1] = PR[90,1] + 69.523;
   1:  PR[91,2] = PR[90,2] + 17.410;
   1:L PR[91] R[100]mm/sec CNT100;
   1:  PR[91,1] = PR[90,1] + 67.660;
   1:  PR[91,2] = PR[90,2] + 16.793;
   1:L PR[91] R[100]mm/sec CNT100;
   1:  PR[91,1] = PR[90,1] + 65.482;
   1:  PR[91,2] = PR[90,2] + 16.108;
   1:L PR[91] R[100]mm/sec CNT100;
   1:  PR[91,1] = PR[90,1] + 64.181;
   1:  PR[91,2] = PR[90,2] + 15.323;
   1:L PR[91] R[100]mm/sec CNT100;
   1:  PR[91,1] = PR[90,1] + 61.820;
   1:  PR[91,2] = PR[90,2] + 13.947;
   1:L PR[91] R[100]mm/sec CNT100;
   1:  PR[91,1] = PR[90,1] + 61.052;
   1:  PR[91,2] = PR[90,2] + 13.205;
   1:L PR[91] R[100]mm/sec CNT100;
   1:  PR[91,1] = PR[90,1] + 58.723;
   1:  PR[91,2] = PR[90,2] + 11.017;
   1:L PR[91] R[100]mm/sec CNT100;
   1:  PR[91,1] = PR[90,1] + 56.378;
   1:  PR[91,2] = PR[90,2] + 7.474;
   1:L PR[91] R[100]mm/sec CNT100;
   1:  PR[91,1] = PR[90,1] + 54.912;
   1:  PR[91,2] = PR[90,2] + 3.488;
   1:L PR[91] R[100]mm/sec CNT100;
   1:  PR[91,1] = PR[90,1] + 54.908;
   1:  PR[91,2] = PR[90,2] + 3.454;
   1:L PR[91] R[100]mm/sec CNT100;
   1:  PR[91,1] = PR[90,1] + 54.425;
   1:  PR[91,2] = PR[90,2] + -0.729;
   1:L PR[91] R[100]mm/sec CNT100;
   1:  PR[91,1] = PR[90,1] + 54.912;
   1:  PR[91,2] = PR[90,2] + -4.949;
   1:L PR[91] R[100]mm/sec CNT100;
   1:  PR[91,1] = PR[90,1] + 56.378;
   1:  PR[91,2] = PR[90,2] + -8.933;
   1:L PR[91] R[100]mm/sec CNT100;
   1:  PR[91,1] = PR[90,1] + 58.730;
   1:  PR[91,2] = PR[90,2] + -12.487;
   1:L PR[91] R[100]mm/sec CNT100;
   1:  PR[91,1] = PR[90,1] + 59.261;
   1:  PR[91,2] = PR[90,2] + -12.998;
   1:L PR[91] R[100]mm/sec CNT100;
   1:  PR[91,1] = PR[90,1] + 61.820;
   1:  PR[91,2] = PR[90,2] + -15.409;
   1:L PR[91] R[100]mm/sec CNT100;
   1:  PR[91,1] = PR[90,1] + 62.881;
   1:  PR[91,2] = PR[90,2] + -16.048;
   1:L PR[91] R[100]mm/sec CNT100;
   1:  PR[91,1] = PR[90,1] + 65.482;
   1:  PR[91,2] = PR[90,2] + -17.571;
   1:L PR[91] R[100]mm/sec CNT100;
   1:  PR[91,1] = PR[90,1] + 67.157;
   1:  PR[91,2] = PR[90,2] + -18.125;
   1:L PR[91] R[100]mm/sec CNT100;
   1:  PR[91,1] = PR[90,1] + 69.522;
   1:  PR[91,2] = PR[90,2] + -18.872;
   1:L PR[91] R[100]mm/sec CNT100;
   1:  PR[91,1] = PR[90,1] + 71.781;
   1:  PR[91,2] = PR[90,2] + -19.095;
   1:L PR[91] R[100]mm/sec CNT100;
   1:  PR[91,1] = PR[90,1] + 73.738;
   1:  PR[91,2] = PR[90,2] + -19.263;
   1:L PR[91] R[100]mm/sec CNT100;
   1:  PR[91,1] = PR[90,1] + 76.433;
   1:  PR[91,2] = PR[90,2] + -18.932;
   1:L PR[91] R[100]mm/sec CNT100;
   1:  PR[91,1] = PR[90,1] + 77.920;
   1:  PR[91,2] = PR[90,2] + -18.731;
   1:L PR[91] R[100]mm/sec CNT100;
   1:  PR[91,1] = PR[90,1] + 80.831;
   1:  PR[91,2] = PR[90,2] + -17.694;
   1:L PR[91] R[100]mm/sec CNT100TB   .50sec,CALL END_PUD;
   1:  PR[92] = PR[91];
   1:  PR[92,3] = PR[92,3] + 20;
   1:J PR[92] 10% FINE;
   1:  PR[91,1] = PR[90,1] + 24.442;
   1:  PR[91,2] = PR[90,2] + 17.762;
   1:  PR[92] = PR[91];
   1:  PR[92,3] = PR[92,3] + 20;
   1:J PR[92] 10% FINE;
   1:L PR[91] R[100]mm/sec CNT100;
   1:  CALL LASER_DRAHT_START;
   1:  PR[91,1] = PR[90,1] + 20.061;
   1:  PR[91,2] = PR[90,2] + 17.192;
   1:L PR[91] R[100]mm/sec CNT100;
   1:  PR[91,1] = PR[90,1] + 19.885;
   1:  PR[91,2] = PR[90,2] + 17.145;
   1:L PR[91] R[100]mm/sec CNT100;
   1:  PR[91,1] = PR[90,1] + 19.558;
   1:  PR[91,2] = PR[90,2] + 16.993;
   1:L PR[91] R[100]mm/sec CNT100;
   1:  PR[91,1] = PR[90,1] + 15.442;
   1:  PR[91,2] = PR[90,2] + 15.297;
   1:L PR[91] R[100]mm/sec CNT100;
   1:  PR[91,1] = PR[90,1] + 15.281;
   1:  PR[91,2] = PR[90,2] + 15.184;
   1:L PR[91] R[100]mm/sec CNT100;
   1:  PR[91,1] = PR[90,1] + 11.695;
   1:  PR[91,2] = PR[90,2] + 12.441;
   1:L PR[91] R[100]mm/sec CNT100;
   1:  PR[91,1] = PR[90,1] + 11.575;
   1:  PR[91,2] = PR[90,2] + 12.322;
   1:L PR[91] R[100]mm/sec CNT100;
   1:  PR[91,1] = PR[90,1] + 8.793;
   1:  PR[91,2] = PR[90,2] + 8.703;
   1:L PR[91] R[100]mm/sec CNT100;
   1:  PR[91,1] = PR[90,1] + 8.683;
   1:  PR[91,2] = PR[90,2] + 8.545;
   1:L PR[91] R[100]mm/sec CNT100;
   1:  PR[91,1] = PR[90,1] + 8.601;
   1:  PR[91,2] = PR[90,2] + 8.370;
   1:L PR[91] R[100]mm/sec CNT100;
   1:  PR[91,1] = PR[90,1] + 6.845;
   1:  PR[91,2] = PR[90,2] + 4.137;
   1:L PR[91] R[100]mm/sec CNT100;
   1:  PR[91,1] = PR[90,1] + 6.821;
   1:  PR[91,2] = PR[90,2] + 4.049;
   1:L PR[91] R[100]mm/sec CNT100;
   1:  PR[91,1] = PR[90,1] + 6.798;
   1:  PR[91,2] = PR[90,2] + 3.785;
   1:L PR[91] R[100]mm/sec CNT100;
   1:  PR[91,1] = PR[90,1] + 6.205;
   1:  PR[91,2] = PR[90,2] + -0.772;
   1:L PR[91] R[100]mm/sec CNT100;
   1:  PR[91,1] = PR[90,1] + 6.232;
   1:  PR[91,2] = PR[90,2] + -1.090;
   1:L PR[91] R[100]mm/sec CNT100;
   1:  PR[91,1] = PR[90,1] + 6.810;
   1:  PR[91,2] = PR[90,2] + -5.465;
   1:L PR[91] R[100]mm/sec CNT100;
   1:  PR[91,1] = PR[90,1] + 6.845;
   1:  PR[91,2] = PR[90,2] + -5.596;
   1:L PR[91] R[100]mm/sec CNT100;
   1:  PR[91,1] = PR[90,1] + 8.601;
   1:  PR[91,2] = PR[90,2] + -9.829;
   1:L PR[91] R[100]mm/sec CNT100;
   1:  PR[91,1] = PR[90,1] + 8.683;
   1:  PR[91,2] = PR[90,2] + -10.004;
   1:L PR[91] R[100]mm/sec CNT100;
   1:  PR[91,1] = PR[90,1] + 8.794;
   1:  PR[91,2] = PR[90,2] + -10.162;
   1:L PR[91] R[100]mm/sec CNT100;
   1:  PR[91,1] = PR[90,1] + 11.576;
   1:  PR[91,2] = PR[90,2] + -13.781;
   1:L PR[91] R[100]mm/sec CNT100;
   1:  PR[91,1] = PR[90,1] + 11.695;
   1:  PR[91,2] = PR[90,2] + -13.900;
   1:L PR[91] R[100]mm/sec CNT100;
   1:  PR[91,1] = PR[90,1] + 15.281;
   1:  PR[91,2] = PR[90,2] + -16.643;
   1:L PR[91] R[100]mm/sec CNT100;
   1:  PR[91,1] = PR[90,1] + 15.480;
   1:  PR[91,2] = PR[90,2] + -16.782;
   1:L PR[91] R[100]mm/sec CNT100;
   1:  PR[91,1] = PR[90,1] + 15.697;
   1:  PR[91,2] = PR[90,2] + -16.883;
   1:L PR[91] R[100]mm/sec CNT100;
   1:  PR[91,1] = PR[90,1] + 19.842;
   1:  PR[91,2] = PR[90,2] + -18.592;
   1:L PR[91] R[100]mm/sec CNT100;
   1:  PR[91,1] = PR[90,1] + 20.063;
   1:  PR[91,2] = PR[90,2] + -18.651;
   1:L PR[91] R[100]mm/sec CNT100;
   1:  PR[91,1] = PR[90,1] + 24.444;
   1:  PR[91,2] = PR[90,2] + -19.221;
   1:L PR[91] R[100]mm/sec CNT100;
   1:  PR[91,1] = PR[90,1] + 24.748;
   1:  PR[91,2] = PR[90,2] + -19.248;
   1:L PR[91] R[100]mm/sec CNT100;
   1:  PR[91,1] = PR[90,1] + 25.049;
   1:  PR[91,2] = PR[90,2] + -19.221;
   1:L PR[91] R[100]mm/sec CNT100;
   1:  PR[91,1] = PR[90,1] + 29.394;
   1:  PR[91,2] = PR[90,2] + -18.641;
   1:L PR[91] R[100]mm/sec CNT100;
   1:  PR[91,1] = PR[90,1] + 29.636;
   1:  PR[91,2] = PR[90,2] + -18.576;
   1:L PR[91] R[100]mm/sec CNT100;
   1:  PR[91,1] = PR[90,1] + 30.018;
   1:  PR[91,2] = PR[90,2] + -18.398;
   1:L PR[91] R[100]mm/sec CNT100;
   1:  PR[91,1] = PR[90,1] + 34.032;
   1:  PR[91,2] = PR[90,2] + -16.727;
   1:L PR[91] R[100]mm/sec CNT100;
   1:  PR[91,1] = PR[90,1] + 34.296;
   1:  PR[91,2] = PR[90,2] + -16.542;
   1:L PR[91] R[100]mm/sec CNT100;
   1:  PR[91,1] = PR[90,1] + 37.698;
   1:  PR[91,2] = PR[90,2] + -13.926;
   1:L PR[91] R[100]mm/sec CNT100;
   1:  PR[91,1] = PR[90,1] + 37.942;
   1:  PR[91,2] = PR[90,2] + -13.682;
   1:L PR[91] R[100]mm/sec CNT100;
   1:  PR[91,1] = PR[90,1] + 40.523;
   1:  PR[91,2] = PR[90,2] + -10.309;
   1:L PR[91] R[100]mm/sec CNT100;
   1:  PR[91,1] = PR[90,1] + 40.759;
   1:  PR[91,2] = PR[90,2] + -9.973;
   1:L PR[91] R[100]mm/sec CNT100;
   1:  PR[91,1] = PR[90,1] + 40.931;
   1:  PR[91,2] = PR[90,2] + -9.604;
   1:L PR[91] R[100]mm/sec CNT100;
   1:  PR[91,1] = PR[90,1] + 42.547;
   1:  PR[91,2] = PR[90,2] + -5.695;
   1:L PR[91] R[100]mm/sec CNT100;
   1:  PR[91,1] = PR[90,1] + 42.634;
   1:  PR[91,2] = PR[90,2] + -5.372;
   1:L PR[91] R[100]mm/sec CNT100;
   1:  PR[91,1] = PR[90,1] + 42.676;
   1:  PR[91,2] = PR[90,2] + -4.882;
   1:L PR[91] R[100]mm/sec CNT100;
   1:  PR[91,1] = PR[90,1] + 43.043;
   1:  PR[91,2] = PR[90,2] + -1.743;
   1:L PR[91] R[100]mm/sec CNT100;
   1:  PR[91,1] = PR[90,1] + 43.191;
   1:  PR[91,2] = PR[90,2] + -0.613;
   1:L PR[91] R[100]mm/sec CNT100;
   1:  PR[91,1] = PR[90,1] + 43.186;
   1:  PR[91,2] = PR[90,2] + -0.242;
   1:L PR[91] R[100]mm/sec CNT100;
   1:  PR[91,1] = PR[90,1] + 42.645;
   1:  PR[91,2] = PR[90,2] + 3.871;
   1:L PR[91] R[100]mm/sec CNT100;
   1:  PR[91,1] = PR[90,1] + 42.547;
   1:  PR[91,2] = PR[90,2] + 4.236;
   1:L PR[91] R[100]mm/sec CNT100;
   1:  PR[91,1] = PR[90,1] + 40.931;
   1:  PR[91,2] = PR[90,2] + 8.145;
   1:L PR[91] R[100]mm/sec CNT100;
   1:  PR[91,1] = PR[90,1] + 40.759;
   1:  PR[91,2] = PR[90,2] + 8.514;
   1:L PR[91] R[100]mm/sec CNT100;
   1:  PR[91,1] = PR[90,1] + 40.523;
   1:  PR[91,2] = PR[90,2] + 8.851;
   1:L PR[91] R[100]mm/sec CNT100;
   1:  PR[91,1] = PR[90,1] + 37.942;
   1:  PR[91,2] = PR[90,2] + 12.223;
   1:L PR[91] R[100]mm/sec CNT100;
   1:  PR[91,1] = PR[90,1] + 37.697;
   1:  PR[91,2] = PR[90,2] + 12.467;
   1:L PR[91] R[100]mm/sec CNT100;
   1:  PR[91,1] = PR[90,1] + 34.296;
   1:  PR[91,2] = PR[90,2] + 15.084;
   1:L PR[91] R[100]mm/sec CNT100;
   1:  PR[91,1] = PR[90,1] + 33.997;
   1:  PR[91,2] = PR[90,2] + 15.293;
   1:L PR[91] R[100]mm/sec CNT100;
   1:  PR[91,1] = PR[90,1] + 33.665;
   1:  PR[91,2] = PR[90,2] + 15.447;
   1:L PR[91] R[100]mm/sec CNT100;
   1:  PR[91,1] = PR[90,1] + 29.676;
   1:  PR[91,2] = PR[90,2] + 17.107;
   1:L PR[91] R[100]mm/sec CNT100;
   1:  PR[91,1] = PR[90,1] + 29.393;
   1:  PR[91,2] = PR[90,2] + 17.183;
   1:L PR[91] R[100]mm/sec CNT100;
   1:  PR[91,1] = PR[90,1] + 25.048;
   1:  PR[91,2] = PR[90,2] + 17.763;
   1:L PR[91] R[100]mm/sec CNT100;
   1:  PR[91,1] = PR[90,1] + 24.747;
   1:  PR[91,2] = PR[90,2] + 17.789;
   1:L PR[91] R[100]mm/sec CNT100;
   1:  PR[91,1] = PR[90,1] + 24.442;
   1:  PR[91,2] = PR[90,2] + 17.762;
   1:L PR[91] R[100]mm/sec CNT100TB   .50sec,CALL END_PUD;
   1:  PR[92] = PR[91];
   1:  PR[92,3] = PR[92,3] + 20;
   1:J PR[92] 10% FINE;
   1:  PR[91,1] = PR[90,1] + -6.135;
   1:  PR[91,2] = PR[90,2] + 2.613;
   1:  PR[92] = PR[91];
   1:  PR[92,3] = PR[92,3] + 20;
   1:J PR[92] 10% FINE;
   1:L PR[91] R[100]mm/sec CNT100;
   1:  CALL LASER_DRAHT_START;
   1:  PR[91,1] = PR[90,1] + -6.132;
   1:  PR[91,2] = PR[90,2] + 2.696;
   1:L PR[91] R[100]mm/sec CNT100;
   1:  PR[91,1] = PR[90,1] + -6.211;
   1:  PR[91,2] = PR[90,2] + 3.378;
   1:L PR[91] R[100]mm/sec CNT100;
   1:  PR[91,1] = PR[90,1] + -7.605;
   1:  PR[91,2] = PR[90,2] + 7.273;
   1:L PR[91] R[100]mm/sec CNT100;
   1:  PR[91,1] = PR[90,1] + -9.848;
   1:  PR[91,2] = PR[90,2] + 10.758;
   1:L PR[91] R[100]mm/sec CNT100;
   1:  PR[91,1] = PR[90,1] + -12.457;
   1:  PR[91,2] = PR[90,2] + 13.307;
   1:L PR[91] R[100]mm/sec CNT100;
   1:  PR[91,1] = PR[90,1] + -12.812;
   1:  PR[91,2] = PR[90,2] + 13.649;
   1:L PR[91] R[100]mm/sec CNT100;
   1:  PR[91,1] = PR[90,1] + -16.362;
   1:  PR[91,2] = PR[90,2] + 15.815;
   1:L PR[91] R[100]mm/sec CNT100;
   1:  PR[91,1] = PR[90,1] + -20.298;
   1:  PR[91,2] = PR[90,2] + 17.139;
   1:L PR[91] R[100]mm/sec CNT100;
   1:  PR[91,1] = PR[90,1] + -24.426;
   1:  PR[91,2] = PR[90,2] + 17.565;
   1:L PR[91] R[100]mm/sec CNT100;
   1:  PR[91,1] = PR[90,1] + -28.515;
   1:  PR[91,2] = PR[90,2] + 17.080;
   1:L PR[91] R[100]mm/sec CNT100;
   1:  PR[91,1] = PR[90,1] + -32.385;
   1:  PR[91,2] = PR[90,2] + 15.719;
   1:L PR[91] R[100]mm/sec CNT100;
   1:  PR[91,1] = PR[90,1] + -35.811;
   1:  PR[91,2] = PR[90,2] + 13.555;
   1:L PR[91] R[100]mm/sec CNT100;
   1:  PR[91,1] = PR[90,1] + -35.829;
   1:  PR[91,2] = PR[90,2] + 13.542;
   1:L PR[91] R[100]mm/sec CNT100;
   1:  PR[91,1] = PR[90,1] + -38.724;
   1:  PR[91,2] = PR[90,2] + 10.635;
   1:L PR[91] R[100]mm/sec CNT100;
   1:  PR[91,1] = PR[90,1] + -38.780;
   1:  PR[91,2] = PR[90,2] + 10.555;
   1:L PR[91] R[100]mm/sec CNT100;
   1:  PR[91,1] = PR[90,1] + -40.861;
   1:  PR[91,2] = PR[90,2] + 7.233;
   1:L PR[91] R[100]mm/sec CNT100;
   1:  PR[91,1] = PR[90,1] + -40.925;
   1:  PR[91,2] = PR[90,2] + 7.096;
   1:L PR[91] R[100]mm/sec CNT100;
   1:  PR[91,1] = PR[90,1] + -42.192;
   1:  PR[91,2] = PR[90,2] + 3.462;
   1:L PR[91] R[100]mm/sec CNT100;
   1:  PR[91,1] = PR[90,1] + -42.239;
   1:  PR[91,2] = PR[90,2] + 3.286;
   1:L PR[91] R[100]mm/sec CNT100;
   1:  PR[91,1] = PR[90,1] + -42.684;
   1:  PR[91,2] = PR[90,2] + -0.752;
   1:L PR[91] R[100]mm/sec CNT100;
   1:  PR[91,1] = PR[90,1] + -42.666;
   1:  PR[91,2] = PR[90,2] + -0.953;
   1:L PR[91] R[100]mm/sec CNT100;
   1:  PR[91,1] = PR[90,1] + -42.240;
   1:  PR[91,2] = PR[90,2] + -4.742;
   1:L PR[91] R[100]mm/sec CNT100;
   1:  PR[91,1] = PR[90,1] + -42.192;
   1:  PR[91,2] = PR[90,2] + -4.921;
   1:L PR[91] R[100]mm/sec CNT100;
   1:  PR[91,1] = PR[90,1] + -40.925;
   1:  PR[91,2] = PR[90,2] + -8.554;
   1:L PR[91] R[100]mm/sec CNT100;
   1:  PR[91,1] = PR[90,1] + -40.861;
   1:  PR[91,2] = PR[90,2] + -8.692;
   1:L PR[91] R[100]mm/sec CNT100;
   1:  PR[91,1] = PR[90,1] + -38.780;
   1:  PR[91,2] = PR[90,2] + -12.014;
   1:L PR[91] R[100]mm/sec CNT100;
   1:  PR[91,1] = PR[90,1] + -38.724;
   1:  PR[91,2] = PR[90,2] + -12.094;
   1:L PR[91] R[100]mm/sec CNT100;
   1:  PR[91,1] = PR[90,1] + -35.829;
   1:  PR[91,2] = PR[90,2] + -15.000;
   1:L PR[91] R[100]mm/sec CNT100;
   1:  PR[91,1] = PR[90,1] + -35.811;
   1:  PR[91,2] = PR[90,2] + -15.013;
   1:L PR[91] R[100]mm/sec CNT100;
   1:  PR[91,1] = PR[90,1] + -32.385;
   1:  PR[91,2] = PR[90,2] + -17.178;
   1:L PR[91] R[100]mm/sec CNT100;
   1:  PR[91,1] = PR[90,1] + -28.515;
   1:  PR[91,2] = PR[90,2] + -18.539;
   1:L PR[91] R[100]mm/sec CNT100;
   1:  PR[91,1] = PR[90,1] + -24.426;
   1:  PR[91,2] = PR[90,2] + -19.024;
   1:L PR[91] R[100]mm/sec CNT100;
   1:  PR[91,1] = PR[90,1] + -20.298;
   1:  PR[91,2] = PR[90,2] + -18.598;
   1:L PR[91] R[100]mm/sec CNT100;
   1:  PR[91,1] = PR[90,1] + -16.362;
   1:  PR[91,2] = PR[90,2] + -17.274;
   1:L PR[91] R[100]mm/sec CNT100;
   1:  PR[91,1] = PR[90,1] + -12.818;
   1:  PR[91,2] = PR[90,2] + -15.111;
   1:L PR[91] R[100]mm/sec CNT100;
   1:  PR[91,1] = PR[90,1] + -9.848;
   1:  PR[91,2] = PR[90,2] + -12.216;
   1:L PR[91] R[100]mm/sec CNT100;
   1:  PR[91,1] = PR[90,1] + -7.605;
   1:  PR[91,2] = PR[90,2] + -8.732;
   1:L PR[91] R[100]mm/sec CNT100;
   1:  PR[91,1] = PR[90,1] + -6.213;
   1:  PR[91,2] = PR[90,2] + -4.840;
   1:L PR[91] R[100]mm/sec CNT100;
   1:  PR[91,1] = PR[90,1] + -5.750;
   1:  PR[91,2] = PR[90,2] + -0.732;
   1:L PR[91] R[100]mm/sec CNT100;
   1:  PR[91,1] = PR[90,1] + -6.135;
   1:  PR[91,2] = PR[90,2] + 2.613;
   1:L PR[91] R[100]mm/sec CNT100TB   .50sec,CALL END_PUD;
   1:  PR[92] = PR[91];
   1:  PR[92,3] = PR[92,3] + 20;
   1:J PR[92] 10% FINE;
   1:  PR[91,1] = PR[90,1] + -88.939;
   1:  PR[91,2] = PR[90,2] + -11.398;
   1:  PR[92] = PR[91];
   1:  PR[92,3] = PR[92,3] + 20;
   1:J PR[92] 10% FINE;
   1:L PR[91] R[100]mm/sec CNT100;
   1:  CALL LASER_DRAHT_START;
   1:  PR[91,1] = PR[90,1] + -86.368;
   1:  PR[91,2] = PR[90,2] + -14.236;
   1:L PR[91] R[100]mm/sec CNT100;
   1:  PR[91,1] = PR[90,1] + -83.249;
   1:  PR[91,2] = PR[90,2] + -16.494;
   1:L PR[91] R[100]mm/sec CNT100;
   1:  PR[91,1] = PR[90,1] + -79.717;
   1:  PR[91,2] = PR[90,2] + -18.073;
   1:L PR[91] R[100]mm/sec CNT100;
   1:  PR[91,1] = PR[90,1] + -75.920;
   1:  PR[91,2] = PR[90,2] + -18.902;
   1:L PR[91] R[100]mm/sec CNT100;
   1:  PR[91,1] = PR[90,1] + -72.026;
   1:  PR[91,2] = PR[90,2] + -18.940;
   1:L PR[91] R[100]mm/sec CNT100;
   1:  PR[91,1] = PR[90,1] + -69.427;
   1:  PR[91,2] = PR[90,2] + -18.416;
   1:L PR[91] R[100]mm/sec CNT100;
   1:  PR[91,1] = PR[90,1] + -68.190;
   1:  PR[91,2] = PR[90,2] + -18.181;
   1:L PR[91] R[100]mm/sec CNT100;
   1:  PR[91,1] = PR[90,1] + -66.042;
   1:  PR[91,2] = PR[90,2] + -17.258;
   1:L PR[91] R[100]mm/sec CNT100;
   1:  PR[91,1] = PR[90,1] + -64.599;
   1:  PR[91,2] = PR[90,2] + -16.655;
   1:L PR[91] R[100]mm/sec CNT100;
   1:  PR[91,1] = PR[90,1] + -62.945;
   1:  PR[91,2] = PR[90,2] + -15.490;
   1:L PR[91] R[100]mm/sec CNT100;
   1:  PR[91,1] = PR[90,1] + -61.397;
   1:  PR[91,2] = PR[90,2] + -14.422;
   1:L PR[91] R[100]mm/sec CNT100;
   1:  PR[91,1] = PR[90,1] + -58.744;
   1:  PR[91,2] = PR[90,2] + -11.582;
   1:L PR[91] R[100]mm/sec CNT100;
   1:  PR[91,1] = PR[90,1] + -56.749;
   1:  PR[91,2] = PR[90,2] + -8.250;
   1:L PR[91] R[100]mm/sec CNT100;
   1:  PR[91,1] = PR[90,1] + -55.514;
   1:  PR[91,2] = PR[90,2] + -4.578;
   1:L PR[91] R[100]mm/sec CNT100;
   1:  PR[91,1] = PR[90,1] + -55.407;
   1:  PR[91,2] = PR[90,2] + -3.591;
   1:L PR[91] R[100]mm/sec CNT100;
   1:  PR[91,1] = PR[90,1] + -55.376;
   1:  PR[91,2] = PR[90,2] + -2.510;
   1:L PR[91] R[100]mm/sec CNT100;
   1:  PR[91,1] = PR[90,1] + -55.203;
   1:  PR[91,2] = PR[90,2] + -0.668;
   1:L PR[91] R[100]mm/sec CNT100;
   1:  PR[91,1] = PR[90,1] + -55.210;
   1:  PR[91,2] = PR[90,2] + -0.437;
   1:L PR[91] R[100]mm/sec CNT100;
   1:  PR[91,1] = PR[90,1] + -55.594;
   1:  PR[91,2] = PR[90,2] + 3.117;
   1:L PR[91] R[100]mm/sec CNT100;
   1:  PR[91,1] = PR[90,1] + -56.822;
   1:  PR[91,2] = PR[90,2] + 6.787;
   1:L PR[91] R[100]mm/sec CNT100;
   1:  PR[91,1] = PR[90,1] + -58.808;
   1:  PR[91,2] = PR[90,2] + 10.117;
   1:L PR[91] R[100]mm/sec CNT100;
   1:  PR[91,1] = PR[90,1] + -61.455;
   1:  PR[91,2] = PR[90,2] + 12.964;
   1:L PR[91] R[100]mm/sec CNT100;
   1:  PR[91,1] = PR[90,1] + -62.398;
   1:  PR[91,2] = PR[90,2] + 13.632;
   1:L PR[91] R[100]mm/sec CNT100;
   1:  PR[91,1] = PR[90,1] + -64.634;
   1:  PR[91,2] = PR[90,2] + 15.192;
   1:L PR[91] R[100]mm/sec CNT100;
   1:  PR[91,1] = PR[90,1] + -68.215;
   1:  PR[91,2] = PR[90,2] + 16.721;
   1:L PR[91] R[100]mm/sec CNT100;
   1:  PR[91,1] = PR[90,1] + -72.030;
   1:  PR[91,2] = PR[90,2] + 17.481;
   1:L PR[91] R[100]mm/sec CNT100;
   1:  PR[91,1] = PR[90,1] + -75.914;
   1:  PR[91,2] = PR[90,2] + 17.445;
   1:L PR[91] R[100]mm/sec CNT100;
   1:  PR[91,1] = PR[90,1] + -79.698;
   1:  PR[91,2] = PR[90,2] + 16.619;
   1:L PR[91] R[100]mm/sec CNT100;
   1:  PR[91,1] = PR[90,1] + -83.220;
   1:  PR[91,2] = PR[90,2] + 15.041;
   1:L PR[91] R[100]mm/sec CNT100;
   1:  PR[91,1] = PR[90,1] + -86.331;
   1:  PR[91,2] = PR[90,2] + 12.784;
   1:L PR[91] R[100]mm/sec CNT100;
   1:  PR[91,1] = PR[90,1] + -88.896;
   1:  PR[91,2] = PR[90,2] + 9.946;
   1:L PR[91] R[100]mm/sec CNT100;
   1:  PR[91,1] = PR[90,1] + -90.810;
   1:  PR[91,2] = PR[90,2] + 6.652;
   1:L PR[91] R[100]mm/sec CNT100;
   1:  PR[91,1] = PR[90,1] + -91.990;
   1:  PR[91,2] = PR[90,2] + 3.041;
   1:L PR[91] R[100]mm/sec CNT100;
   1:  PR[91,1] = PR[90,1] + -92.373;
   1:  PR[91,2] = PR[90,2] + -0.547;
   1:L PR[91] R[100]mm/sec CNT100;
   1:  PR[91,1] = PR[90,1] + -92.432;
   1:  PR[91,2] = PR[90,2] + -0.831;
   1:L PR[91] R[100]mm/sec CNT100;
